C07299=1229.702,-97.800,-36.392,179.567,5.287,149.048
C07300=1229.707,-98.050,-36.382,179.565,5.287,149.049
C07301=1229.712,-98.299,-36.370,179.563,5.287,149.049
C07302=1229.718,-98.549,-36.360,179.561,5.287,149.050
C07303=1229.723,-98.799,-36.350,179.558,5.287,149.051
C07304=1229.728,-99.048,-36.339,179.556,5.287,149.052
C07305=1229.733,-99.298,-36.328,179.553,5.286,149.052
C07306=1229.738,-99.548,-36.318,179.551,5.287,149.053
C07307=1229.743,-99.798,-36.307,179.548,5.286,149.054
C07308=1229.748,-100.048,-36.296,179.546,5.287,149.054
C07309=1229.755,-100.319,-36.285,179.544,5.286,149.055
C07310=1229.759,-100.589,-36.273,179.542,5.287,149.056
C07311=1229.765,-100.861,-36.262,179.538,5.287,149.057
C07312=1229.772,-101.131,-36.250,179.536,5.286,149.057
C07313=1229.777,-101.382,-36.239,179.534,5.287,149.058
C07314=1229.782,-101.631,-36.229,179.531,5.286,149.059
C07315=1229.787,-101.881,-36.218,179.529,5.286,149.060
C07316=1229.793,-102.130,-36.207,179.527,5.286,149.060
C07317=1229.797,-102.380,-36.197,179.525,5.286,149.061
C07318=1229.802,-102.630,-36.187,179.523,5.286,149.062
C07319=1229.807,-102.880,-36.177,179.520,5.286,149.062
C07320=1229.813,-103.129,-36.166,179.518,5.286,149.063
C07321=1229.818,-103.379,-36.155,179.515,5.286,149.064
C07322=1229.823,-103.629,-36.145,179.513,5.286,149.064
C07323=1229.828,-103.879,-36.134,179.510,5.286,149.065
C07324=1229.834,-104.129,-36.124,179.508,5.286,149.066
C07325=1229.839,-104.377,-36.113,179.506,5.286,149.067
C07326=1229.844,-104.628,-36.103,179.503,5.286,149.067
C07327=1229.850,-104.877,-36.092,179.501,5.286,149.068
C07328=1229.855,-105.127,-36.082,179.499,5.286,149.069
C07329=1229.860,-105.377,-36.072,179.496,5.286,149.069
C07330=1229.865,-105.627,-36.061,179.494,5.286,149.070
C07331=1229.870,-105.876,-36.051,179.492,5.285,149.071
C07332=1229.875,-106.126,-36.040,179.490,5.285,149.071
C07333=1229.880,-106.376,-36.030,179.487,5.285,149.072
C07334=1229.886,-106.625,-36.020,179.485,5.285,149.073
C07335=1229.891,-106.875,-36.009,179.483,5.286,149.073
C07336=1229.897,-107.125,-35.999,179.480,5.285,149.074
C07337=1229.902,-107.375,-35.988,179.478,5.286,149.075
C07338=1229.907,-107.625,-35.978,179.475,5.285,149.076
C07339=1229.913,-107.874,-35.968,179.473,5.286,149.076
C07340=1229.917,-108.124,-35.957,179.471,5.285,149.077
C07341=1229.922,-108.373,-35.947,179.468,5.286,149.078
C07342=1229.927,-108.623,-35.937,179.466,5.285,149.078
C07343=1229.933,-108.873,-35.926,179.464,5.285,149.079
C07344=1229.939,-109.123,-35.916,179.462,5.285,149.080
C07345=1229.944,-109.373,-35.906,179.459,5.285,149.080
C07346=1229.948,-109.622,-35.896,179.457,5.285,149.081
C07347=1229.953,-109.872,-35.885,179.455,5.285,149.082
C07348=1229.959,-110.122,-35.875,179.453,5.285,149.082
C07349=1229.965,-110.371,-35.865,179.450,5.285,149.083
C07350=1229.970,-110.622,-35.854,179.448,5.285,149.084
C07351=1229.975,-110.871,-35.845,179.445,5.285,149.085
C07352=1229.980,-111.120,-35.835,179.443,5.285,149.085
C07353=1229.985,-111.371,-35.824,179.441,5.284,149.086
C07354=1229.991,-111.620,-35.814,179.439,5.285,149.087
C07355=1229.996,-111.870,-35.804,179.436,5.284,149.087
C07356=1230.001,-112.120,-35.794,179.434,5.285,149.088
C07357=1230.006,-112.369,-35.783,179.431,5.284,149.089
C07358=1230.011,-112.619,-35.773,179.429,5.285,149.089
C07359=1230.017,-112.869,-35.763,179.427,5.284,149.090
C07360=1230.022,-113.118,-35.752,179.424,5.285,149.091
C07361=1230.027,-113.368,-35.742,179.422,5.285,149.092
C07362=1230.032,-113.618,-35.732,179.420,5.285,149.092
C07363=1230.038,-113.867,-35.722,179.418,5.285,149.093
C07364=1230.044,-114.118,-35.712,179.415,5.284,149.093
C07365=1230.048,-114.368,-35.702,179.413,5.284,149.094
C07366=1230.054,-114.617,-35.692,179.411,5.284,149.095
C07367=1230.059,-114.867,-35.682,179.409,5.284,149.096
C07368=1230.064,-115.117,-35.671,179.406,5.284,149.096
C07369=1230.069,-115.366,-35.662,179.404,5.284,149.097
C07370=1230.075,-115.616,-35.652,179.401,5.284,149.098
C07371=1230.080,-115.866,-35.641,179.399,5.284,149.098
C07372=1230.085,-116.115,-35.631,179.397,5.284,149.099
C07373=1230.090,-116.365,-35.622,179.395,5.284,149.100
C07374=1230.095,-116.616,-35.611,179.393,5.284,149.100
C07375=1230.100,-116.865,-35.602,179.390,5.284,149.101
C07376=1230.106,-117.114,-35.592,179.388,5.284,149.102
C07377=1230.111,-117.364,-35.581,179.385,5.284,149.103
C07378=1230.116,-117.614,-35.571,179.383,5.284,149.103
C07379=1230.122,-117.864,-35.562,179.380,5.284,149.104
C07380=1230.127,-118.114,-35.552,179.379,5.284,149.104
C07381=1230.132,-118.363,-35.542,179.376,5.283,149.105
C07382=1230.137,-118.613,-35.532,179.374,5.284,149.106
C07383=1230.143,-118.863,-35.521,179.372,5.284,149.107
C07384=1230.148,-119.112,-35.512,179.369,5.284,149.107
C07385=1230.153,-119.363,-35.502,179.367,5.284,149.108
C07386=1230.158,-119.612,-35.492,179.364,5.284,149.109
C07387=1230.163,-119.861,-35.482,179.362,5.284,149.109
C07388=1230.169,-120.111,-35.472,179.360,5.283,149.110
C07389=1230.174,-120.362,-35.462,179.358,5.283,149.111
C07390=1230.179,-120.611,-35.452,179.355,5.283,149.111
C07391=1230.185,-120.861,-35.442,179.353,5.283,149.112
C07392=1230.190,-121.110,-35.433,179.351,5.284,149.113
C07393=1230.195,-121.360,-35.423,179.349,5.283,149.114
C07394=1230.200,-121.610,-35.412,179.346,5.284,149.114
C07395=1230.205,-121.859,-35.403,179.344,5.283,149.115
C07396=1230.211,-122.110,-35.393,179.342,5.283,149.115
C07397=1230.216,-122.359,-35.384,179.339,5.283,149.116
C07398=1230.221,-122.609,-35.373,179.337,5.283,149.117
C07399=1230.226,-122.859,-35.364,179.335,5.283,149.118
C07400=1230.232,-123.109,-35.354,179.333,5.283,149.118
C07401=1230.237,-123.358,-35.344,179.331,5.284,149.119
C07402=1230.243,-123.608,-35.335,179.328,5.283,149.120
C07403=1230.248,-123.858,-35.324,179.326,5.283,149.120
C07404=1230.252,-124.107,-35.315,179.324,5.283,149.121
C07405=1230.258,-124.358,-35.305,179.321,5.283,149.122
C07406=1230.263,-124.607,-35.296,179.319,5.283,149.122
C07407=1230.269,-124.856,-35.285,179.317,5.283,149.123
C07408=1230.273,-125.107,-35.276,179.314,5.283,149.124
C07409=1230.279,-125.356,-35.266,179.312,5.283,149.125
C07410=1230.284,-125.606,-35.256,179.310,5.283,149.125
C07411=1230.290,-125.856,-35.247,179.308,5.283,149.126
C07412=1230.295,-126.105,-35.237,179.306,5.283,149.126
C07413=1229.874,-126.116,-35.273,179.301,5.287,149.129
C07414=1229.868,-125.866,-35.282,179.303,5.286,149.128
C07415=1229.863,-125.617,-35.292,179.305,5.286,149.127
C07416=1229.857,-125.367,-35.302,179.308,5.286,149.126
C07417=1229.852,-125.117,-35.311,179.310,5.286,149.126
C07418=1229.846,-124.868,-35.321,179.313,5.286,149.125
C07419=1229.842,-124.617,-35.331,179.314,5.286,149.125
C07420=1229.836,-124.368,-35.341,179.317,5.287,149.124
C07421=1229.831,-124.118,-35.351,179.319,5.286,149.123
C07422=1229.826,-123.868,-35.360,179.322,5.287,149.122
C07423=1229.821,-123.619,-35.370,179.324,5.286,149.122
C07424=1229.816,-123.369,-35.380,179.326,5.286,149.121
C07425=1229.810,-123.119,-35.389,179.328,5.287,149.120
C07426=1229.805,-122.869,-35.399,179.330,5.286,149.120
C07427=1229.799,-122.620,-35.409,179.333,5.287,149.119
C07428=1229.794,-122.370,-35.418,179.335,5.286,149.118
C07429=1229.789,-122.120,-35.429,179.338,5.287,149.118
C07430=1229.784,-121.871,-35.439,179.340,5.286,149.117
C07431=1229.778,-121.620,-35.448,179.342,5.287,149.116
C07432=1229.773,-121.371,-35.458,179.345,5.287,149.115
C07433=1229.769,-121.121,-35.468,179.346,5.287,149.115
C07434=1229.763,-120.871,-35.478,179.349,5.287,149.114
C07435=1229.758,-120.622,-35.487,179.351,5.287,149.114
C07436=1229.752,-120.372,-35.498,179.354,5.287,149.113
C07437=1229.747,-120.122,-35.508,179.356,5.287,149.112
C07438=1229.742,-119.872,-35.518,179.358,5.287,149.111
C07439=1229.736,-119.622,-35.527,179.360,5.287,149.111
C07440=1229.732,-119.373,-35.537,179.363,5.287,149.110
C07441=1229.726,-119.124,-35.547,179.365,5.287,149.109
C07442=1229.721,-118.873,-35.558,179.367,5.288,149.109
C07443=1229.716,-118.623,-35.567,179.370,5.287,149.108
C07444=1229.710,-118.374,-35.577,179.372,5.287,149.107
C07445=1229.705,-118.124,-35.587,179.374,5.287,149.107
C07446=1229.700,-117.874,-35.597,179.376,5.287,149.106
C07447=1229.695,-117.625,-35.607,179.379,5.287,149.105
C07448=1229.689,-117.375,-35.617,179.381,5.287,149.105
C07449=1229.685,-117.125,-35.627,179.383,5.288,149.104
C07450=1229.679,-116.875,-35.637,179.385,5.287,149.103
C07451=1229.673,-116.626,-35.647,179.388,5.288,149.103
C07452=1229.668,-116.376,-35.657,179.390,5.287,149.102
C07453=1229.663,-116.126,-35.667,179.393,5.288,149.101
C07454=1229.658,-115.877,-35.677,179.395,5.287,149.100
C07455=1229.653,-115.627,-35.686,179.397,5.287,149.100
C07456=1229.648,-115.377,-35.697,179.399,5.288,149.099
C07457=1229.642,-115.127,-35.707,179.401,5.287,149.098
C07458=1229.637,-114.878,-35.717,179.404,5.288,149.098
C07459=1229.632,-114.628,-35.727,179.406,5.288,149.097
C07460=1229.627,-114.378,-35.738,179.409,5.288,149.096
C07461=1229.621,-114.128,-35.748,179.411,5.288,149.096
C07462=1229.616,-113.878,-35.758,179.414,5.288,149.095
C07463=1229.611,-113.629,-35.768,179.416,5.288,149.094
C07464=1229.606,-113.379,-35.778,179.418,5.288,149.093
C07465=1229.600,-113.129,-35.788,179.420,5.288,149.093
C07466=1229.595,-112.879,-35.798,179.422,5.288,149.092
C07467=1229.590,-112.630,-35.808,179.425,5.288,149.092
C07468=1229.584,-112.380,-35.818,179.427,5.288,149.091
C07469=1229.579,-112.130,-35.829,179.430,5.288,149.090
C07470=1229.574,-111.880,-35.839,179.432,5.288,149.089
C07471=1229.569,-111.631,-35.849,179.434,5.288,149.089
C07472=1229.564,-111.381,-35.859,179.436,5.288,149.088
C07473=1229.558,-111.131,-35.869,179.439,5.288,149.087
C07474=1229.553,-110.881,-35.880,179.441,5.288,149.087
C07475=1229.548,-110.632,-35.890,179.443,5.289,149.086
C07476=1229.543,-110.382,-35.900,179.445,5.288,149.085
C07477=1229.538,-110.132,-35.910,179.448,5.288,149.085
C07478=1229.532,-109.883,-35.920,179.450,5.288,149.084
C07479=1229.527,-109.633,-35.931,179.452,5.288,149.083
C07480=1229.522,-109.383,-35.941,179.455,5.289,149.082
C07481=1229.517,-109.134,-35.951,179.457,5.288,149.082
C07482=1229.512,-108.883,-35.961,179.460,5.289,149.081
C07483=1229.506,-108.634,-35.972,179.462,5.288,149.080
C07484=1229.500,-108.384,-35.982,179.465,5.289,149.080
C07485=1229.496,-108.135,-35.993,179.467,5.288,149.079
C07486=1229.490,-107.885,-36.003,179.469,5.289,149.078
C07487=1229.485,-107.635,-36.014,179.471,5.289,149.078
C07488=1229.480,-107.386,-36.023,179.474,5.289,149.077
C07489=1229.475,-107.136,-36.034,179.476,5.289,149.076
C07490=1229.470,-106.886,-36.044,179.478,5.289,149.076
C07491=1229.464,-106.636,-36.054,179.480,5.289,149.075
C07492=1229.459,-106.386,-36.065,179.483,5.289,149.074
C07493=1229.454,-106.137,-36.075,179.485,5.289,149.073
C07494=1229.448,-105.887,-36.085,179.487,5.289,149.073
C07495=1229.443,-105.637,-36.097,179.490,5.289,149.072
C07496=1229.438,-105.388,-36.106,179.492,5.289,149.071
C07497=1229.433,-105.138,-36.117,179.495,5.289,149.071
C07498=1229.428,-104.888,-36.127,179.496,5.289,149.070
C07499=1229.423,-104.638,-36.138,179.499,5.290,149.069
C07500=1229.417,-104.389,-36.148,179.501,5.289,149.069
C07501=1229.413,-104.139,-36.159,179.504,5.290,149.068
C07502=1229.407,-103.889,-36.169,179.506,5.289,149.067
C07503=1229.401,-103.640,-36.180,179.509,5.290,149.066
C07504=1229.396,-103.390,-36.190,179.511,5.289,149.066
C07505=1229.391,-103.140,-36.200,179.513,5.290,149.065
C07506=1229.386,-102.890,-36.212,179.515,5.289,149.064
C07507=1229.380,-102.641,-36.222,179.517,5.289,149.064
C07508=1229.375,-102.391,-36.232,179.520,5.289,149.063
C07509=1229.370,-102.141,-36.243,179.522,5.289,149.062
C07510=1229.365,-101.891,-36.253,179.525,5.290,149.062
C07511=1229.360,-101.642,-36.264,179.527,5.290,149.061
C07512=1229.355,-101.392,-36.275,179.529,5.290,149.060
C07513=1229.350,-101.142,-36.284,179.531,5.290,149.060
C07514=1229.344,-100.871,-36.297,179.534,5.290,149.059
C07515=1229.338,-100.600,-36.308,179.537,5.290,149.058
C07516=1229.333,-100.330,-36.319,179.539,5.290,149.057
C07517=1229.327,-100.058,-36.331,179.542,5.290,149.057
C07518=1229.322,-99.808,-36.342,179.544,5.290,149.056
C07519=1229.316,-99.559,-36.352,179.547,5.290,149.055
C07520=1229.311,-99.309,-36.363,179.549,5.290,149.054
C07521=1229.306,-99.059,-36.373,179.551,5.290,149.054
C07522=1229.301,-98.810,-36.385,179.554,5.290,149.053
C07523=1229.296,-98.560,-36.395,179.556,5.290,149.052
C07524=1229.291,-98.310,-36.405,179.558,5.290,149.052
C07525=1229.285,-98.061,-36.416,179.561,5.291,149.051
C07526=1229.280,-97.811,-36.427,179.563,5.291,149.050
C07527=1229.275,-97.561,-36.437,179.565,5.290,149.050
C07528=1229.270,-97.312,-36.448,179.567,5.291,149.049
C07529=1229.264,-97.062,-36.459,179.569,5.290,149.048
C07530=1229.259,-96.812,-36.469,179.572,5.291,149.047
C07531=1229.254,-96.563,-36.480,179.574,5.290,149.047
C07532=1229.249,-96.313,-36.491,179.577,5.291,149.046
C07533=1229.243,-96.063,-36.501,179.579,5.290,149.045
C07534=1229.238,-95.813,-36.513,179.582,5.291,149.045
C07535=1229.233,-95.563,-36.523,179.584,5.291,149.044
C07536=1229.228,-95.314,-36.534,179.586,5.291,149.043
C07537=1229.223,-95.064,-36.545,179.589,5.291,149.042
C07538=1229.218,-94.815,-36.556,179.591,5.291,149.042
C07539=1229.213,-94.565,-36.566,179.593,5.291,149.041
C07540=1229.207,-94.315,-36.576,179.596,5.291,149.040
C07541=1229.202,-94.065,-36.588,179.598,5.291,149.040
C07542=1229.196,-93.815,-36.599,179.601,5.291,149.039
C07543=1229.191,-93.566,-36.610,179.603,5.291,149.038
C07544=1229.186,-93.316,-36.620,179.606,5.291,149.037
C07545=1229.181,-93.067,-36.631,179.607,5.291,149.037
C07546=1229.176,-92.817,-36.642,179.610,5.292,149.036
C07547=1229.171,-92.567,-36.653,179.612,5.291,149.036
C07548=1229.166,-92.317,-36.663,179.615,5.292,149.035
C07549=1229.160,-92.067,-36.675,179.617,5.292,149.034
C07550=1229.155,-91.818,-36.686,179.619,5.292,149.033
C07551=1229.150,-91.568,-36.697,179.621,5.292,149.033
C07552=1229.145,-91.318,-36.707,179.624,5.292,149.032
C07553=1229.140,-91.069,-36.718,179.626,5.292,149.031
C07554=1229.135,-90.819,-36.729,179.629,5.292,149.031
C07555=1229.129,-90.570,-36.740,179.631,5.292,149.030
C07556=1229.124,-90.319,-36.751,179.634,5.292,149.029
C07557=1229.119,-90.070,-36.762,179.636,5.292,149.028
C07558=1229.114,-89.821,-36.773,179.638,5.292,149.028
C07559=1229.109,-89.571,-36.784,179.640,5.292,149.027
C07560=1229.103,-89.321,-36.796,179.643,5.292,149.026
C07561=1229.098,-89.071,-36.806,179.645,5.292,149.026
C07562=1229.093,-88.821,-36.817,179.648,5.293,149.025
C07563=1229.088,-88.571,-36.828,179.650,5.292,149.024
C07564=1229.082,-88.322,-36.839,179.653,5.293,149.023
C07565=1229.077,-88.072,-36.851,179.655,5.292,149.023
C07566=1229.072,-87.822,-36.861,179.657,5.293,149.022
C07567=1229.067,-87.573,-36.872,179.660,5.292,149.021
C07568=1229.061,-87.323,-36.884,179.662,5.293,149.021
C07569=1229.056,-87.073,-36.895,179.664,5.292,149.020
C07570=1229.051,-86.824,-36.905,179.666,5.293,149.019
C07571=1229.046,-86.574,-36.917,179.669,5.293,149.019
C07572=1229.041,-86.324,-36.928,179.671,5.293,149.018
C07573=1229.035,-86.075,-36.939,179.673,5.293,149.017
C07574=1229.031,-85.825,-36.950,179.675,5.293,149.017
C07575=1229.025,-85.575,-36.961,179.678,5.293,149.016
C07576=1229.020,-85.326,-36.972,179.680,5.293,149.015
C07577=1229.015,-85.076,-36.983,179.683,5.293,149.014
C07578=1229.010,-84.826,-36.994,179.686,5.294,149.014
C07579=1229.005,-84.576,-37.006,179.688,5.293,149.013
C07580=1228.999,-84.327,-37.017,179.690,5.294,149.012
C07581=1228.994,-84.077,-37.027,179.692,5.293,149.012
C07582=1228.989,-83.827,-37.039,179.695,5.294,149.011
C07583=1228.984,-83.578,-37.050,179.697,5.294,149.010
C07584=1228.979,-83.328,-37.062,179.700,5.294,149.010
C07585=1228.973,-83.078,-37.073,179.702,5.294,149.009
C07586=1228.968,-82.828,-37.084,179.705,5.294,149.008
C07587=1228.963,-82.579,-37.095,179.707,5.294,149.007
C07588=1228.958,-82.329,-37.107,179.709,5.294,149.007
C07589=1228.953,-82.080,-37.118,179.711,5.294,149.006
C07590=1228.948,-81.829,-37.129,179.714,5.294,149.005
C07591=1228.942,-81.580,-37.140,179.716,5.294,149.005
C07592=1228.937,-81.331,-37.151,179.719,5.294,149.004
C07593=1228.932,-81.081,-37.163,179.721,5.294,149.003
C07594=1228.927,-80.831,-37.175,179.724,5.295,149.002
C07595=1228.922,-80.582,-37.185,179.726,5.294,149.002
C07596=1228.916,-80.332,-37.197,179.728,5.295,149.001
C07597=1228.911,-80.082,-37.208,179.730,5.294,149.000
C07598=1228.906,-79.832,-37.220,179.733,5.295,149.000
C07599=1228.901,-79.583,-37.231,179.735,5.294,148.999
C07600=1228.896,-79.333,-37.242,179.738,5.295,148.998
C07601=1228.890,-79.083,-37.253,179.740,5.295,148.997
C07602=1228.886,-78.833,-37.265,179.743,5.295,148.997
C07603=1228.880,-78.583,-37.277,179.745,5.295,148.996
C07604=1228.875,-78.334,-37.287,179.747,5.295,148.995
C07605=1228.869,-78.084,-37.299,179.750,5.295,148.995
C07606=1228.865,-77.835,-37.311,179.752,5.295,148.994
C07607=1228.860,-77.585,-37.322,179.754,5.295,148.993
C07608=1228.855,-77.335,-37.334,179.757,5.295,148.992
C07609=1228.849,-77.086,-37.345,179.759,5.295,148.992
C07610=1228.844,-76.836,-37.356,179.762,5.295,148.991
C07611=1228.839,-76.586,-37.367,179.764,5.295,148.990
C07612=1228.834,-76.336,-37.379,179.766,5.296,148.990
C07613=1228.829,-76.087,-37.390,179.769,5.295,148.989
C07614=1228.823,-75.837,-37.402,179.771,5.296,148.988
C07615=1228.818,-75.588,-37.413,179.773,5.295,148.988
C07616=1228.813,-75.338,-37.425,179.776,5.296,148.987
C07617=1228.808,-75.088,-37.436,179.778,5.295,148.986
C07618=1228.802,-74.819,-37.449,179.781,5.296,148.985
C07619=1228.796,-74.548,-37.461,179.783,5.296,148.985
C07620=1228.791,-74.277,-37.474,179.786,5.296,148.984
C07621=1228.785,-74.007,-37.486,179.788,5.296,148.983
C07622=1228.780,-73.757,-37.498,179.791,5.297,148.983
C07623=1228.775,-73.507,-37.509,179.793,5.297,148.982
C07624=1228.769,-73.257,-37.521,179.796,5.297,148.981
C07625=1228.765,-73.008,-37.533,179.798,5.297,148.980
C07626=1228.760,-72.759,-37.545,179.800,5.297,148.980
C07627=1228.755,-72.509,-37.556,179.802,5.297,148.979
C07628=1228.749,-72.260,-37.568,179.805,5.297,148.978
C07629=1228.744,-72.010,-37.579,179.807,5.297,148.978
C07630=1228.739,-71.760,-37.591,179.810,5.297,148.977
C07631=1228.733,-71.510,-37.603,179.812,5.297,148.976
C07632=1228.729,-71.261,-37.614,179.815,5.298,148.975
C07633=1228.723,-71.011,-37.626,179.817,5.297,148.975
C07634=1228.718,-70.761,-37.637,179.819,5.298,148.974
C07635=1228.713,-70.511,-37.649,179.822,5.297,148.973
C07636=1228.707,-70.262,-37.661,179.824,5.298,148.973
C07637=1228.702,-70.012,-37.672,179.826,5.297,148.972
C07638=1228.697,-69.763,-37.685,179.829,5.298,148.971
C07639=1228.693,-69.513,-37.696,179.832,5.298,148.971
C07640=1228.687,-69.263,-37.708,179.834,5.298,148.970
C07641=1228.682,-69.013,-37.720,179.836,5.298,148.969
C07642=1228.677,-68.764,-37.731,179.838,5.298,148.968
C07643=1228.672,-68.514,-37.743,179.841,5.299,148.968
C07644=1228.666,-68.264,-37.755,179.843,5.298,148.967
C07645=1228.662,-68.015,-37.767,179.846,5.299,148.966
C07646=1228.656,-67.765,-37.779,179.848,5.298,148.966
C07647=1228.651,-67.515,-37.790,179.851,5.299,148.965
C07648=1228.646,-67.266,-37.801,179.853,5.299,148.964
C07649=1228.640,-67.016,-37.813,179.855,5.299,148.963
C07650=1228.635,-66.767,-37.826,179.858,5.299,148.963
C07651=1228.630,-66.517,-37.837,179.860,5.299,148.962
C07652=1228.625,-66.267,-37.849,179.862,5.299,148.961
C07653=1228.619,-66.017,-37.861,179.865,5.299,148.961
C07654=1228.615,-65.768,-37.872,179.868,5.300,148.960
C07655=1228.610,-65.518,-37.885,179.870,5.299,148.959
C07656=1228.604,-65.268,-37.897,179.872,5.300,148.959
C07657=1228.600,-65.019,-37.908,179.874,5.300,148.958
C07658=1228.594,-64.769,-37.920,179.877,5.300,148.957
C07659=1228.589,-64.520,-37.933,179.879,5.300,148.956
C07660=1228.584,-64.270,-37.944,179.882,5.300,148.956
C07661=1228.579,-64.020,-37.956,179.884,5.300,148.955
C07662=1228.574,-63.771,-37.968,179.887,5.300,148.954
C07663=1228.568,-63.521,-37.980,179.889,5.300,148.954
C07664=1228.564,-63.271,-37.991,179.891,5.300,148.953
C07665=1228.558,-63.022,-38.004,179.894,5.301,148.952
C07666=1228.553,-62.772,-38.016,179.897,5.300,148.951
C07667=1228.548,-62.522,-38.028,179.899,5.301,148.951
C07668=1228.543,-62.273,-38.040,179.901,5.300,148.950
C07669=1228.538,-62.023,-38.052,179.904,5.301,148.949
C07670=1228.532,-61.773,-38.064,179.906,5.300,148.948
C07671=1228.527,-61.524,-38.076,179.909,5.301,148.948
C07672=1228.522,-61.274,-38.088,179.911,5.301,148.947
C07673=1228.517,-61.024,-38.099,179.914,5.301,148.946
C07674=1228.512,-60.775,-38.112,179.916,5.301,148.946
C07675=1228.507,-60.525,-38.124,179.918,5.301,148.945
C07676=1228.501,-60.275,-38.136,179.921,5.302,148.944
C07677=1228.496,-60.026,-38.148,179.923,5.301,148.943
C07678=1228.491,-59.776,-38.160,179.926,5.302,148.943
C07679=1228.486,-59.527,-38.172,179.928,5.301,148.942
C07680=1228.481,-59.277,-38.184,179.931,5.302,148.941
C07681=1228.476,-59.027,-38.197,179.933,5.302,148.941
C07682=1228.470,-58.777,-38.209,179.935,5.302,148.940
C07683=1228.466,-58.528,-38.220,179.937,5.302,148.939
C07684=1228.461,-58.278,-38.233,179.940,5.302,148.939
C07685=1228.456,-58.028,-38.245,179.943,5.303,148.938
C07686=1228.450,-57.779,-38.257,179.945,5.302,148.937
C07687=1228.445,-57.529,-38.269,179.947,5.303,148.936
C07688=1228.440,-57.279,-38.282,179.950,5.302,148.936
C07689=1228.434,-57.029,-38.294,179.952,5.303,148.935
C07690=1228.430,-56.780,-38.306,179.954,5.303,148.934
C07691=1228.425,-56.530,-38.318,179.957,5.303,148.934
C07692=1228.420,-56.281,-38.330,179.960,5.304,148.933
C07693=1228.414,-56.031,-38.342,179.962,5.303,148.932
C07694=1228.409,-55.782,-38.355,179.964,5.304,148.931
C07695=1228.404,-55.532,-38.367,179.966,5.303,148.931
C07696=1228.399,-55.282,-38.380,179.969,5.304,148.930
C07697=1228.394,-55.032,-38.391,179.971,5.304,148.929
C07698=1228.388,-54.783,-38.404,179.974,5.304,148.929
C07699=1228.384,-54.534,-38.416,179.976,5.304,148.928
C07700=1228.379,-54.284,-38.428,179.979,5.304,148.927
C07701=1228.374,-54.034,-38.441,179.981,5.305,148.927
C07702=1228.368,-53.784,-38.452,179.983,5.304,148.926
C07703=1228.363,-53.535,-38.465,179.986,5.305,148.925
C07704=1228.358,-53.285,-38.477,179.988,5.304,148.924
C07705=1228.353,-53.035,-38.490,179.991,5.305,148.924
C07706=1228.348,-52.786,-38.502,179.993,5.305,148.923
C07707=1228.342,-52.536,-38.514,179.996,5.305,148.922
C07708=1228.337,-52.287,-38.527,179.998,5.306,148.922
C07709=1228.332,-52.037,-38.540,-180.000,5.305,148.921
C07710=1228.327,-51.787,-38.551,-179.997,5.306,148.920
C07711=1228.322,-51.537,-38.564,-179.995,5.305,148.920
C07712=1228.317,-51.287,-38.576,-179.992,5.306,148.919
C07713=1228.312,-51.038,-38.589,-179.990,5.306,148.918
C07714=1228.307,-50.789,-38.602,-179.988,5.306,148.917
C07715=1228.301,-50.539,-38.613,-179.985,5.306,148.917
C07716=1228.296,-50.290,-38.626,-179.983,5.306,148.916
C07717=1228.292,-50.040,-38.639,-179.980,5.307,148.915
C07718=1228.286,-49.790,-38.651,-179.978,5.306,148.915
C07719=1228.281,-49.540,-38.663,-179.975,5.307,148.914
C07720=1228.276,-49.291,-38.676,-179.973,5.307,148.913
C07721=1228.271,-49.042,-38.689,-179.971,5.307,148.912
C07722=1228.265,-48.771,-38.702,-179.967,5.307,148.912
C07723=1228.260,-48.501,-38.716,-179.965,5.308,148.911
C07724=1228.254,-48.232,-38.729,-179.963,5.307,148.910
C07725=1228.249,-47.962,-38.742,-179.960,5.308,148.909
C07726=1228.244,-47.713,-38.755,-179.957,5.308,148.909
C07727=1228.239,-47.463,-38.767,-179.955,5.308,148.908
C07728=1228.234,-47.213,-38.780,-179.953,5.308,148.907
C07729=1228.229,-46.963,-38.792,-179.951,5.308,148.907
C07730=1228.223,-46.714,-38.805,-179.948,5.309,148.906
C07731=1228.218,-46.464,-38.818,-179.946,5.308,148.905
C07732=1228.212,-46.215,-38.831,-179.943,5.308,148.904
C07733=1228.208,-45.965,-38.844,-179.940,5.309,148.904
C07734=1228.203,-45.715,-38.855,-179.938,5.308,148.903
C07735=1228.197,-45.466,-38.868,-179.935,5.309,148.902
C07736=1228.192,-45.216,-38.881,-179.933,5.309,148.901
C07737=1228.188,-44.966,-38.894,-179.930,5.309,148.901
C07738=1228.183,-44.717,-38.906,-179.928,5.310,148.900
C07739=1228.177,-44.467,-38.919,-179.926,5.309,148.899
C07740=1228.171,-44.218,-38.931,-179.923,5.310,148.899
C07741=1228.167,-43.967,-38.944,-179.921,5.309,148.898
C07742=1228.162,-43.718,-38.957,-179.918,5.310,148.897
C07743=1228.157,-43.469,-38.969,-179.916,5.310,148.897
C07744=1228.151,-43.220,-38.982,-179.914,5.310,148.896
C07745=1228.147,-42.970,-38.995,-179.911,5.311,148.895
C07746=1228.141,-42.720,-39.008,-179.909,5.310,148.894
C07747=1228.136,-42.471,-39.021,-179.906,5.311,148.894
C07748=1228.131,-42.221,-39.034,-179.903,5.311,148.893
C07749=1228.126,-41.971,-39.046,-179.901,5.311,148.892
C07750=1228.121,-41.721,-39.058,-179.899,5.311,148.892
C07751=1228.116,-41.472,-39.071,-179.897,5.311,148.891
C07752=1228.110,-41.222,-39.084,-179.894,5.312,148.890
C07753=1228.105,-40.972,-39.097,-179.891,5.312,148.890
C07754=1228.100,-40.723,-39.110,-179.889,5.312,148.889
C07755=1228.096,-40.473,-39.123,-179.887,5.312,148.888
C07756=1228.090,-40.223,-39.136,-179.884,5.312,148.887
C07757=1228.085,-39.974,-39.148,-179.882,5.312,148.887
C07758=1228.080,-39.724,-39.161,-179.879,5.313,148.886
C07759=1228.075,-39.475,-39.174,-179.877,5.313,148.885
C07760=1228.070,-39.225,-39.187,-179.874,5.313,148.885
C07761=1228.064,-38.976,-39.200,-179.872,5.313,148.884
C07762=1228.060,-38.726,-39.213,-179.870,5.313,148.883
C07763=1228.054,-38.476,-39.225,-179.867,5.314,148.883
C07764=1228.049,-38.227,-39.238,-179.865,5.313,148.882
C07765=1228.044,-37.977,-39.252,-179.862,5.314,148.881
C07766=1228.039,-37.727,-39.264,-179.860,5.314,148.880
C07767=1228.034,-37.478,-39.277,-179.857,5.314,148.880
C07768=1228.029,-37.228,-39.290,-179.855,5.315,148.879
C07769=1228.023,-36.979,-39.303,-179.853,5.314,148.878
C07770=1228.019,-36.728,-39.316,-179.850,5.315,148.878
C07771=1228.014,-36.480,-39.329,-179.847,5.315,148.877
C07772=1228.008,-36.230,-39.342,-179.845,5.315,148.876
C07773=1228.004,-35.980,-39.355,-179.843,5.315,148.876
C07774=1227.999,-35.731,-39.368,-179.841,5.315,148.875
C07775=1227.993,-35.481,-39.381,-179.838,5.316,148.874
C07776=1227.988,-35.231,-39.394,-179.835,5.316,148.873
C07777=1227.983,-34.982,-39.407,-179.833,5.315,148.873
C07778=1227.977,-34.732,-39.420,-179.830,5.316,148.872
C07779=1227.973,-34.482,-39.433,-179.828,5.316,148.871
C07780=1227.968,-34.234,-39.446,-179.825,5.316,148.870
C07781=1227.963,-33.983,-39.460,-179.823,5.317,148.870
C07782=1227.957,-33.734,-39.472,-179.821,5.316,148.869
C07783=1227.952,-33.485,-39.485,-179.818,5.317,148.868
C07784=1227.947,-33.234,-39.499,-179.815,5.317,148.868
C07785=1227.942,-32.985,-39.511,-179.813,5.317,148.867
C07786=1227.937,-32.735,-39.525,-179.810,5.317,148.866
C07787=1227.932,-32.486,-39.538,-179.808,5.317,148.866
C07788=1227.927,-32.236,-39.551,-179.806,5.318,148.865
C07789=1227.921,-31.986,-39.564,-179.803,5.318,148.864
C07790=1227.917,-31.738,-39.577,-179.801,5.318,148.863
C07791=1227.911,-31.487,-39.591,-179.798,5.318,148.863
C07792=1227.906,-31.238,-39.604,-179.796,5.319,148.862
C07793=1227.902,-30.988,-39.617,-179.794,5.318,148.861
C07794=1227.896,-30.738,-39.630,-179.791,5.319,148.861
C07795=1227.892,-30.489,-39.643,-179.789,5.319,148.860
C07796=1227.886,-30.239,-39.657,-179.786,5.319,148.859
C07797=1227.881,-29.990,-39.669,-179.783,5.320,148.859
C07798=1227.876,-29.741,-39.683,-179.781,5.319,148.858
C07799=1227.871,-29.491,-39.696,-179.779,5.320,148.857
C07800=1227.866,-29.241,-39.709,-179.776,5.320,148.856
C07801=1227.860,-28.991,-39.722,-179.774,5.320,148.856
C07802=1227.856,-28.742,-39.736,-179.771,5.321,148.855
C07803=1227.850,-28.492,-39.749,-179.769,5.321,148.854
C07804=1227.846,-28.242,-39.762,-179.767,5.321,148.854
C07805=1227.840,-27.993,-39.776,-179.764,5.321,148.853
C07806=1227.836,-27.743,-39.789,-179.762,5.321,148.852
C07807=1227.830,-27.494,-39.802,-179.759,5.321,148.852
C07808=1227.825,-27.244,-39.816,-179.757,5.322,148.851
C07809=1227.820,-26.994,-39.829,-179.754,5.322,148.850
C07810=1227.815,-26.745,-39.843,-179.752,5.322,148.849
C07811=1227.810,-26.495,-39.856,-179.749,5.323,148.849
C07812=1227.805,-26.245,-39.869,-179.747,5.322,148.848
C07813=1227.799,-25.996,-39.883,-179.744,5.323,148.847
C07814=1227.795,-25.746,-39.896,-179.742,5.323,148.847
C07815=1227.789,-25.497,-39.909,-179.740,5.323,148.846
C07816=1227.785,-25.247,-39.923,-179.737,5.323,148.845
C07817=1227.779,-24.998,-39.936,-179.734,5.324,148.845
C07818=1227.775,-24.748,-39.950,-179.732,5.324,148.844
C07819=1227.769,-24.499,-39.963,-179.730,5.324,148.843
C07820=1227.765,-24.249,-39.976,-179.727,5.325,148.843
C07821=1227.759,-24.000,-39.990,-179.725,5.324,148.842
C07822=1227.754,-23.750,-40.004,-179.722,5.325,148.841
C07823=1227.749,-23.501,-40.017,-179.719,5.325,148.840
C07824=1227.744,-23.251,-40.031,-179.717,5.325,148.840
C07825=1227.739,-23.001,-40.044,-179.714,5.325,148.839
C07826=1227.733,-22.732,-40.058,-179.712,5.326,148.838
C07827=1227.728,-22.463,-40.073,-179.710,5.325,148.837
C07828=1227.723,-22.193,-40.087,-179.707,5.326,148.837
C07829=1227.717,-21.924,-40.102,-179.704,5.326,148.836
C07830=1227.712,-21.675,-40.116,-179.701,5.327,148.835
C07831=1227.707,-21.425,-40.129,-179.699,5.326,148.834
C07832=1227.702,-21.176,-40.143,-179.696,5.327,148.834
C07833=1227.696,-20.925,-40.156,-179.694,5.327,148.833
C07834=1227.692,-20.677,-40.170,-179.692,5.327,148.832
C07835=1227.686,-20.426,-40.183,-179.689,5.327,148.832
C07836=1227.681,-20.177,-40.198,-179.686,5.328,148.831
C07837=1227.676,-19.927,-40.210,-179.684,5.328,148.830
C07838=1227.671,-19.678,-40.224,-179.682,5.328,148.830
C07839=1227.666,-19.429,-40.238,-179.679,5.329,148.829
C07840=1227.661,-19.179,-40.251,-179.677,5.328,148.828
C07841=1227.656,-18.929,-40.266,-179.674,5.329,148.827
C07842=1227.650,-18.679,-40.279,-179.671,5.329,148.827
C07843=1227.646,-18.430,-40.292,-179.669,5.329,148.826
C07844=1227.641,-18.181,-40.306,-179.667,5.330,148.825
C07845=1227.635,-17.930,-40.320,-179.664,5.330,148.825
C07846=1227.631,-17.681,-40.334,-179.662,5.330,148.824
C07847=1227.626,-17.432,-40.348,-179.659,5.330,148.823
C07848=1227.620,-17.182,-40.361,-179.657,5.331,148.823
C07849=1227.615,-16.933,-40.375,-179.655,5.330,148.822
C07850=1227.611,-16.683,-40.389,-179.652,5.331,148.821
C07851=1227.605,-16.433,-40.402,-179.649,5.332,148.821
C07852=1227.600,-16.184,-40.416,-179.647,5.331,148.820
C07853=1227.596,-15.935,-40.430,-179.645,5.332,148.819
C07854=1227.590,-15.684,-40.443,-179.642,5.332,148.818
C07855=1227.585,-15.435,-40.457,-179.640,5.332,148.818
C07856=1227.580,-15.186,-40.472,-179.637,5.332,148.817
C07857=1227.576,-14.936,-40.485,-179.635,5.333,148.816
C07858=1227.570,-14.686,-40.498,-179.632,5.333,148.816
C07859=1227.565,-14.437,-40.513,-179.630,5.333,148.815
C07860=1227.560,-14.187,-40.527,-179.627,5.334,148.814
C07861=1227.554,-13.938,-40.541,-179.625,5.333,148.814
C07862=1227.550,-13.688,-40.554,-179.622,5.334,148.813
C07863=1227.545,-13.438,-40.568,-179.620,5.334,148.812
C07864=1227.539,-13.189,-40.582,-179.617,5.335,148.811
C07865=1227.534,-12.940,-40.596,-179.615,5.335,148.811
C07866=1227.530,-12.690,-40.609,-179.612,5.335,148.810
C07867=1227.524,-12.441,-40.623,-179.610,5.336,148.809
C07868=1227.519,-12.191,-40.638,-179.608,5.335,148.809
C07869=1227.514,-11.941,-40.652,-179.605,5.336,148.808
C07870=1227.509,-11.691,-40.666,-179.602,5.336,148.807
C07871=1227.504,-11.442,-40.679,-179.600,5.336,148.807
C07872=1227.499,-11.192,-40.693,-179.598,5.337,148.806
C07873=1227.494,-10.943,-40.707,-179.595,5.337,148.805
C07874=1227.489,-10.694,-40.721,-179.593,5.337,148.805
C07875=1227.484,-10.444,-40.735,-179.590,5.337,148.804
C07876=1227.479,-10.194,-40.750,-179.587,5.338,148.803
C07877=1227.474,-9.945,-40.764,-179.585,5.338,148.802
C07878=1227.468,-9.696,-40.778,-179.583,5.338,148.802
C07879=1227.464,-9.446,-40.791,-179.580,5.339,148.801
C07880=1227.459,-9.196,-40.805,-179.577,5.339,148.800
C07881=1227.454,-8.946,-40.819,-179.575,5.339,148.800
C07882=1227.448,-8.697,-40.833,-179.573,5.339,148.799
C07883=1227.443,-8.447,-40.848,-179.570,5.340,148.798
C07884=1227.438,-8.198,-40.862,-179.568,5.340,148.798
C07885=1227.434,-7.948,-40.876,-179.565,5.340,148.797
C07886=1227.428,-7.699,-40.890,-179.563,5.341,148.796
C07887=1227.423,-7.449,-40.904,-179.560,5.341,148.796
C07888=1227.419,-7.200,-40.918,-179.558,5.341,148.795
C07889=1227.414,-6.950,-40.932,-179.555,5.341,148.794
C07890=1227.409,-6.700,-40.947,-179.553,5.342,148.793
C07891=1227.403,-6.451,-40.961,-179.551,5.342,148.793
C07892=1227.398,-6.202,-40.975,-179.548,5.342,148.792
C07893=1227.393,-5.952,-40.989,-179.545,5.343,148.791
C07894=1227.388,-5.702,-41.003,-179.543,5.343,148.791
C07895=1227.383,-5.453,-41.018,-179.541,5.343,148.790
C07896=1227.378,-5.204,-41.032,-179.538,5.343,148.789
C07897=1227.373,-4.954,-41.046,-179.535,5.344,148.789
C07898=1227.368,-4.704,-41.060,-179.533,5.344,148.788
C07899=1227.363,-4.454,-41.074,-179.530,5.344,148.787
C07900=1227.358,-4.205,-41.089,-179.528,5.345,148.787
C07901=1227.353,-3.956,-41.103,-179.525,5.345,148.786
C07902=1227.348,-3.706,-41.117,-179.523,5.345,148.785
C07903=1227.343,-3.456,-41.131,-179.520,5.345,148.785
C07904=1227.338,-3.207,-41.145,-179.518,5.346,148.784
C07905=1227.333,-2.957,-41.160,-179.516,5.346,148.783
C07906=1227.328,-2.707,-41.174,-179.513,5.346,148.782
C07907=1227.323,-2.459,-41.189,-179.510,5.347,148.782
C07908=1227.318,-2.209,-41.203,-179.508,5.347,148.781
C07909=1227.313,-1.959,-41.217,-179.506,5.347,148.780
C07910=1227.308,-1.710,-41.231,-179.503,5.347,148.780
C07911=1227.303,-1.460,-41.246,-179.500,5.348,148.779
C07912=1227.298,-1.210,-41.260,-179.498,5.348,148.778
C07913=1227.292,-0.961,-41.274,-179.496,5.348,148.778
C07914=1227.288,-0.712,-41.289,-179.493,5.349,148.777
C07915=1227.283,-0.462,-41.303,-179.490,5.349,148.776
C07916=1227.278,-0.213,-41.317,-179.488,5.349,148.776
C07917=1227.272,0.037,-41.332,-179.486,5.349,148.775
C07918=1227.267,0.287,-41.347,-179.483,5.350,148.774
C07919=1227.262,0.537,-41.361,-179.480,5.350,148.773
C07920=1227.257,0.786,-41.376,-179.478,5.350,148.773
C07921=1227.252,1.035,-41.390,-179.476,5.351,148.772
C07922=1227.247,1.285,-41.404,-179.473,5.351,148.771
C07923=1227.242,1.534,-41.418,-179.470,5.352,148.771
C07924=1227.237,1.783,-41.433,-179.468,5.351,148.770
C07925=1227.232,2.033,-41.448,-179.466,5.352,148.769
C07926=1227.227,2.283,-41.462,-179.463,5.352,148.769
C07927=1227.222,2.533,-41.477,-179.460,5.353,148.768
C07928=1227.217,2.782,-41.492,-179.458,5.353,148.767
C07929=1227.212,3.032,-41.506,-179.455,5.353,148.767
C07930=1227.207,3.300,-41.522,-179.453,5.354,148.766
C07931=1227.202,3.569,-41.537,-179.450,5.354,148.765
C07932=1227.195,3.838,-41.553,-179.447,5.354,148.764
C07933=1227.190,4.107,-41.568,-179.444,5.355,148.764
C07934=1227.185,4.356,-41.583,-179.442,5.355,148.763
C07935=1227.180,4.606,-41.598,-179.440,5.355,148.762
C07936=1227.175,4.856,-41.612,-179.437,5.356,148.762
C07937=1227.170,5.105,-41.627,-179.434,5.356,148.761
C07938=1227.165,5.355,-41.642,-179.432,5.356,148.760
C07939=1227.160,5.604,-41.656,-179.430,5.357,148.759
C07940=1227.155,5.853,-41.671,-179.427,5.357,148.759
C07941=1227.150,6.103,-41.685,-179.424,5.358,148.758
C07942=1227.145,6.353,-41.700,-179.422,5.357,148.757
C07943=1227.140,6.602,-41.715,-179.420,5.358,148.757
C07944=1227.135,6.852,-41.729,-179.417,5.358,148.756
C07945=1227.131,7.101,-41.744,-179.414,5.359,148.755
C07946=1227.125,7.351,-41.759,-179.412,5.359,148.755
C07947=1227.120,7.601,-41.774,-179.410,5.359,148.754
C07948=1227.115,7.850,-41.789,-179.407,5.360,148.753
C07949=1227.110,8.100,-41.803,-179.404,5.360,148.753
C07950=1227.105,8.349,-41.818,-179.402,5.360,148.752
C07951=1227.100,8.599,-41.833,-179.400,5.360,148.751
C07952=1227.095,8.848,-41.848,-179.397,5.361,148.751
C07953=1227.090,9.098,-41.862,-179.394,5.361,148.750
C07954=1227.085,9.347,-41.878,-179.392,5.362,148.749
C07955=1227.080,9.597,-41.892,-179.389,5.362,148.748
C07956=1227.075,9.846,-41.907,-179.387,5.362,148.748
C07957=1227.070,10.096,-41.922,-179.384,5.363,148.747
C07958=1227.065,10.345,-41.937,-179.382,5.363,148.746
C07959=1227.060,10.595,-41.951,-179.379,5.363,148.746
C07960=1227.055,10.844,-41.967,-179.377,5.364,148.745
C07961=1227.050,11.094,-41.981,-179.374,5.364,148.744
C07962=1227.045,11.343,-41.996,-179.372,5.365,148.744
C07963=1227.039,11.593,-42.011,-179.370,5.365,148.743
C07964=1227.035,11.842,-42.026,-179.367,5.365,148.743
C07965=1227.030,12.092,-42.040,-179.365,5.366,148.742
C07966=1227.024,12.341,-42.056,-179.362,5.366,148.741
C07967=1227.019,12.591,-42.070,-179.359,5.367,148.741
C07968=1227.015,12.840,-42.085,-179.357,5.367,148.740
C07969=1227.009,13.089,-42.100,-179.355,5.367,148.739
C07970=1227.005,13.340,-42.115,-179.352,5.368,148.738
C07971=1227.000,13.589,-42.130,-179.349,5.368,148.738
C07972=1226.995,13.838,-42.146,-179.347,5.369,148.737
C07973=1226.990,14.088,-42.160,-179.345,5.368,148.736
C07974=1226.985,14.337,-42.176,-179.342,5.369,148.736
C07975=1226.980,14.587,-42.190,-179.339,5.370,148.735
C07976=1226.975,14.836,-42.205,-179.337,5.370,148.734
C07977=1226.970,15.085,-42.220,-179.335,5.370,148.734
C07978=1226.965,15.335,-42.235,-179.332,5.370,148.733
C07979=1226.959,15.585,-42.250,-179.329,5.371,148.732
C07980=1226.955,15.834,-42.265,-179.327,5.371,148.732
C07981=1226.949,16.084,-42.280,-179.324,5.372,148.731
C07982=1226.945,16.333,-42.295,-179.322,5.372,148.730
C07983=1226.940,16.583,-42.310,-179.319,5.372,148.730
C07984=1226.935,16.832,-42.326,-179.317,5.373,148.729
C07985=1226.930,17.082,-42.340,-179.314,5.373,148.728
C07986=1226.925,17.331,-42.356,-179.311,5.374,148.728
C07987=1226.920,17.580,-42.371,-179.309,5.374,148.727
C07988=1226.914,17.830,-42.386,-179.307,5.374,148.726
C07989=1226.910,18.079,-42.401,-179.304,5.375,148.725
C07990=1226.905,18.329,-42.417,-179.301,5.375,148.725
C07991=1226.900,18.578,-42.432,-179.299,5.376,148.724
C07992=1226.895,18.828,-42.447,-179.297,5.375,148.723
C07993=1226.890,19.078,-42.462,-179.294,5.376,148.723
C07994=1226.884,19.327,-42.477,-179.292,5.377,148.722
C07995=1226.880,19.576,-42.492,-179.289,5.377,148.722
C07996=1226.875,19.826,-42.508,-179.286,5.378,148.721
C07997=1226.870,20.075,-42.523,-179.284,5.378,148.720
C07998=1226.865,20.325,-42.538,-179.282,5.378,148.720
C07999=1226.860,20.574,-42.553,-179.279,5.379,148.719
C08000=1226.855,20.824,-42.569,-179.276,5.379,148.718
C08001=1226.850,21.073,-42.584,-179.274,5.380,148.718
C08002=1226.845,21.323,-42.599,-179.271,5.380,148.717
C08003=1226.840,21.572,-42.615,-179.269,5.380,148.716
C08004=1226.835,21.822,-42.629,-179.266,5.381,148.715
C08005=1226.829,22.071,-42.645,-179.264,5.381,148.715
C08006=1226.825,22.321,-42.660,-179.261,5.382,148.714
C08007=1226.820,22.571,-42.676,-179.259,5.382,148.713
C08008=1226.815,22.820,-42.691,-179.256,5.382,148.713
C08009=1226.810,23.069,-42.706,-179.254,5.383,148.712
C08010=1226.805,23.319,-42.722,-179.251,5.383,148.711
C08011=1226.800,23.568,-42.737,-179.249,5.384,148.711
C08012=1226.795,23.818,-42.753,-179.246,5.384,148.710
C08013=1226.790,24.067,-42.768,-179.243,5.385,148.709
C08014=1226.785,24.316,-42.784,-179.242,5.385,148.709
C08015=1226.780,24.566,-42.799,-179.239,5.385,148.708
C08016=1226.776,24.815,-42.815,-179.236,5.386,148.708
C08017=1226.770,25.065,-42.830,-179.234,5.386,148.707
C08018=1226.765,25.314,-42.846,-179.231,5.387,148.706
C08019=1226.760,25.563,-42.861,-179.228,5.388,148.705
C08020=1226.755,25.813,-42.877,-179.226,5.387,148.705
C08021=1226.750,26.063,-42.892,-179.224,5.388,148.704
C08022=1226.745,26.312,-42.907,-179.221,5.388,148.703
C08023=1226.740,26.561,-42.923,-179.218,5.389,148.703
C08024=1226.735,26.811,-42.939,-179.216,5.389,148.702
C08025=1226.731,27.061,-42.954,-179.213,5.390,148.701
C08026=1226.725,27.310,-42.969,-179.211,5.390,148.701
C08027=1226.720,27.559,-42.985,-179.208,5.390,148.700
C08028=1226.716,27.809,-43.000,-179.206,5.391,148.699
C08029=1226.710,28.059,-43.016,-179.203,5.391,148.699
C08030=1226.705,28.308,-43.031,-179.200,5.392,148.698
C08031=1226.701,28.558,-43.047,-179.198,5.393,148.698
C08032=1226.696,28.807,-43.062,-179.196,5.393,148.697
C08033=1226.690,29.057,-43.078,-179.194,5.393,148.696
C08034=1226.685,29.325,-43.095,-179.191,5.394,148.696
C08035=1226.680,29.593,-43.111,-179.188,5.394,148.695
C08036=1226.675,29.862,-43.129,-179.185,5.394,148.694
C08037=1226.669,30.131,-43.146,-179.183,5.395,148.693
C08038=1226.664,30.380,-43.161,-179.180,5.395,148.693
C08039=1226.659,30.630,-43.177,-179.177,5.396,148.692
C08040=1226.654,30.879,-43.192,-179.175,5.397,148.691
C08041=1226.649,31.129,-43.208,-179.172,5.397,148.691
C08042=1226.644,31.378,-43.224,-179.169,5.398,148.690
C08043=1226.639,31.628,-43.240,-179.167,5.397,148.689
C08044=1226.634,31.877,-43.256,-179.165,5.398,148.689
C08045=1226.629,32.126,-43.271,-179.162,5.399,148.688
C08046=1226.624,32.376,-43.287,-179.160,5.399,148.687
C08047=1226.619,32.626,-43.302,-179.157,5.400,148.687
C08048=1226.615,32.875,-43.319,-179.155,5.401,148.686
C08049=1226.609,33.125,-43.335,-179.152,5.401,148.685
C08050=1226.604,33.374,-43.350,-179.150,5.401,148.685
C08051=1226.600,33.624,-43.366,-179.147,5.401,148.684
C08052=1226.595,33.873,-43.382,-179.145,5.402,148.683
C08053=1226.589,34.122,-43.397,-179.142,5.402,148.683
C08054=1226.584,34.372,-43.413,-179.139,5.403,148.682
C08055=1226.579,34.621,-43.430,-179.137,5.404,148.681
C08056=1226.575,34.871,-43.445,-179.134,5.404,148.681
C08057=1226.570,35.120,-43.461,-179.132,5.404,148.680
C08058=1226.565,35.369,-43.476,-179.130,5.405,148.679
C08059=1226.560,35.619,-43.493,-179.127,5.405,148.679
C08060=1226.555,35.868,-43.509,-179.124,5.406,148.678
C08061=1226.549,36.118,-43.524,-179.122,5.406,148.677
C08062=1226.545,36.367,-43.541,-179.119,5.407,148.677
C08063=1226.539,36.617,-43.556,-179.117,5.408,148.676
C08064=1226.535,36.867,-43.572,-179.114,5.408,148.675
C08065=1226.530,37.115,-43.588,-179.112,5.408,148.675
C08066=1226.526,37.365,-43.604,-179.109,5.408,148.674
C08067=1226.520,37.614,-43.620,-179.107,5.409,148.673
C08068=1226.515,37.863,-43.636,-179.104,5.410,148.673
C08069=1226.510,38.114,-43.652,-179.102,5.410,148.672
C08070=1226.505,38.362,-43.668,-179.099,5.411,148.672
C08071=1226.500,38.612,-43.684,-179.096,5.412,148.671
C08072=1226.495,38.861,-43.700,-179.094,5.412,148.670
C08073=1226.491,39.111,-43.716,-179.091,5.413,148.670
C08074=1226.485,39.361,-43.732,-179.089,5.412,148.669
C08075=1226.480,39.610,-43.748,-179.086,5.413,148.668
C08076=1226.475,39.860,-43.764,-179.084,5.413,148.668
C08077=1226.470,40.108,-43.780,-179.081,5.414,148.667
C08078=1226.465,40.359,-43.796,-179.079,5.415,148.666
C08079=1226.460,40.607,-43.813,-179.076,5.416,148.666
C08080=1226.456,40.857,-43.829,-179.074,5.416,148.665
C08081=1226.450,41.106,-43.845,-179.071,5.417,148.664
C08082=1226.446,41.356,-43.861,-179.068,5.417,148.664
C08083=1226.441,41.605,-43.877,-179.066,5.418,148.663
C08084=1226.436,41.855,-43.893,-179.064,5.418,148.662
C08085=1226.431,42.104,-43.909,-179.061,5.418,148.662
C08086=1226.426,42.354,-43.925,-179.058,5.419,148.661
C08087=1226.421,42.603,-43.942,-179.056,5.419,148.660
C08088=1226.416,42.852,-43.958,-179.053,5.420,148.660
C08089=1226.411,43.102,-43.974,-179.051,5.421,148.659
C08090=1226.407,43.351,-43.991,-179.048,5.421,148.659
C08091=1226.401,43.601,-44.006,-179.046,5.422,148.658
C08092=1226.397,43.850,-44.023,-179.043,5.422,148.657
C08093=1226.391,44.100,-44.039,-179.041,5.423,148.657
C08094=1226.386,44.349,-44.056,-179.038,5.423,148.656
C08095=1226.381,44.598,-44.072,-179.036,5.423,148.655
C08096=1226.376,44.848,-44.088,-179.033,5.424,148.655
C08097=1226.371,45.097,-44.104,-179.031,5.424,148.654
C08098=1226.367,45.346,-44.121,-179.028,5.425,148.653
C08099=1226.362,45.597,-44.137,-179.026,5.426,148.653
C08100=1226.357,45.845,-44.153,-179.023,5.426,148.652
C08101=1226.352,46.095,-44.169,-179.020,5.427,148.651
C08102=1226.347,46.344,-44.186,-179.018,5.428,148.651
C08103=1226.342,46.594,-44.203,-179.015,5.428,148.650
C08104=1226.337,46.843,-44.219,-179.013,5.429,148.649
C08105=1226.332,47.093,-44.235,-179.010,5.429,148.649
C08106=1226.327,47.342,-44.251,-179.008,5.430,148.648
C08107=1226.322,47.591,-44.268,-179.006,5.430,148.648
C08108=1226.317,47.841,-44.284,-179.003,5.430,148.647
C08109=1226.312,48.090,-44.300,-179.000,5.431,148.646
C08110=1226.307,48.340,-44.318,-178.998,5.432,148.646
C08111=1226.302,48.589,-44.334,-178.995,5.432,148.645
C08112=1226.297,48.839,-44.350,-178.993,5.433,148.644
C08113=1226.293,49.088,-44.366,-178.990,5.433,148.644
C08114=1226.288,49.337,-44.383,-178.988,5.434,148.643
C08115=1226.282,49.587,-44.400,-178.985,5.435,148.642
C08116=1226.277,49.836,-44.416,-178.982,5.435,148.642
C08117=1226.273,50.086,-44.432,-178.980,5.436,148.641
C08118=1226.268,50.335,-44.449,-178.977,5.436,148.640
C08119=1226.263,50.584,-44.465,-178.975,5.437,148.640
C08120=1226.258,50.834,-44.483,-178.972,5.438,148.639
C08121=1226.253,51.083,-44.499,-178.969,5.438,148.638
C08122=1226.248,51.333,-44.515,-178.968,5.438,148.638
C08123=1226.243,51.582,-44.531,-178.965,5.439,148.637
C08124=1226.238,51.831,-44.548,-178.962,5.439,148.637
C08125=1226.233,52.081,-44.565,-178.960,5.440,148.636
C08126=1226.229,52.330,-44.582,-178.957,5.441,148.635
C08127=1226.224,52.579,-44.598,-178.955,5.441,148.635
C08128=1226.218,52.829,-44.615,-178.952,5.442,148.634
C08129=1226.214,53.079,-44.631,-178.950,5.443,148.634
C08130=1226.209,53.328,-44.648,-178.947,5.443,148.633
C08131=1226.204,53.577,-44.664,-178.944,5.444,148.632
C08132=1226.199,53.827,-44.681,-178.942,5.444,148.632
C08133=1226.194,54.076,-44.698,-178.939,5.445,148.631
C08134=1226.189,54.325,-44.714,-178.937,5.445,148.630
C08135=1226.184,54.575,-44.732,-178.934,5.446,148.630
C08136=1226.179,54.824,-44.748,-178.932,5.447,148.629
C08137=1226.175,55.073,-44.765,-178.929,5.447,148.628
C08138=1226.169,55.342,-44.783,-178.927,5.448,148.628
C08139=1226.164,55.610,-44.801,-178.924,5.449,148.627
C08140=1226.158,55.880,-44.819,-178.921,5.449,148.626
C08141=1226.153,56.147,-44.837,-178.918,5.449,148.626
C08142=1226.148,56.397,-44.853,-178.916,5.450,148.625
C08143=1226.143,56.647,-44.871,-178.913,5.451,148.624
C08144=1226.138,56.895,-44.887,-178.911,5.451,148.624
C08145=1226.134,57.145,-44.904,-178.908,5.452,148.623
C08146=1226.128,57.395,-44.921,-178.905,5.453,148.622
C08147=1226.123,57.643,-44.937,-178.903,5.453,148.622
C08148=1226.118,57.893,-44.955,-178.900,5.454,148.621
C08149=1226.114,58.142,-44.972,-178.898,5.455,148.621
C08150=1226.110,58.392,-44.989,-178.895,5.455,148.620
C08151=1226.104,58.641,-45.005,-178.893,5.456,148.619
C08152=1226.099,58.890,-45.022,-178.890,5.456,148.619
C08153=1226.094,59.140,-45.039,-178.887,5.457,148.618
C08154=1226.090,59.389,-45.056,-178.885,5.458,148.617
C08155=1226.084,59.639,-45.073,-178.883,5.459,148.617
C08156=1226.079,59.888,-45.090,-178.880,5.459,148.616
C08157=1226.074,60.138,-45.107,-178.877,5.460,148.616
C08158=1226.070,60.387,-45.124,-178.875,5.460,148.615
C08159=1226.065,60.636,-45.141,-178.872,5.461,148.614
C08160=1226.060,60.885,-45.158,-178.870,5.461,148.614
C08161=1226.055,61.135,-45.175,-178.867,5.462,148.613
C08162=1226.050,61.385,-45.192,-178.865,5.463,148.612
C08163=1226.045,61.634,-45.208,-178.862,5.463,148.612
C08164=1226.040,61.883,-45.226,-178.860,5.464,148.611
C08165=1226.035,62.132,-45.243,-178.857,5.465,148.610
C08166=1226.030,62.382,-45.260,-178.854,5.465,148.610
C08167=1226.026,62.631,-45.277,-178.852,5.466,148.609
C08168=1226.020,62.881,-45.294,-178.849,5.467,148.609
C08169=1226.016,63.129,-45.311,-178.847,5.467,148.608
C08170=1226.010,63.379,-45.328,-178.844,5.468,148.607
C08171=1226.006,63.629,-45.345,-178.842,5.468,148.607
C08172=1226.001,63.878,-45.362,-178.839,5.469,148.606
C08173=1225.997,64.127,-45.380,-178.837,5.470,148.606
C08174=1225.991,64.377,-45.397,-178.834,5.471,148.605
C08175=1225.986,64.626,-45.414,-178.832,5.471,148.604
C08176=1225.981,64.875,-45.431,-178.829,5.472,148.604
C08177=1225.976,65.125,-45.448,-178.826,5.472,148.603
C08178=1225.972,65.374,-45.465,-178.824,5.473,148.603
C08179=1225.967,65.623,-45.483,-178.822,5.474,148.602
C08180=1225.962,65.873,-45.500,-178.819,5.474,148.601
C08181=1225.956,66.122,-45.517,-178.816,5.475,148.601
C08182=1225.952,66.371,-45.535,-178.814,5.476,148.600
C08183=1225.947,66.621,-45.551,-178.811,5.476,148.599
C08184=1225.942,66.870,-45.569,-178.809,5.477,148.599
C08185=1225.938,67.119,-45.586,-178.806,5.478,148.598
C08186=1225.932,67.369,-45.603,-178.804,5.478,148.597
C08187=1225.927,67.619,-45.620,-178.801,5.479,148.597
C08188=1225.923,67.868,-45.638,-178.798,5.479,148.596
C08189=1225.917,68.117,-45.655,-178.796,5.480,148.596
C08190=1225.912,68.366,-45.673,-178.794,5.481,148.595
C08191=1225.908,68.616,-45.689,-178.791,5.481,148.594
C08192=1225.903,68.865,-45.707,-178.788,5.482,148.594
C08193=1225.898,69.114,-45.725,-178.786,5.483,148.593
C08194=1225.893,69.364,-45.741,-178.784,5.484,148.593
C08195=1225.888,69.613,-45.759,-178.781,5.484,148.592
C08196=1225.883,69.863,-45.777,-178.778,5.485,148.591
C08197=1225.879,70.112,-45.794,-178.776,5.485,148.591
C08198=1225.874,70.362,-45.811,-178.773,5.486,148.590
C08199=1225.869,70.611,-45.829,-178.771,5.487,148.590
C08200=1225.864,70.860,-45.846,-178.768,5.487,148.589
C08201=1225.859,71.109,-45.863,-178.766,5.488,148.588
C08202=1225.854,71.359,-45.881,-178.763,5.489,148.588
C08203=1225.849,71.607,-45.898,-178.761,5.489,148.587
C08204=1225.844,71.857,-45.915,-178.758,5.491,148.586
C08205=1225.839,72.106,-45.933,-178.755,5.491,148.586
C08206=1225.834,72.356,-45.951,-178.752,5.492,148.585
C08207=1225.830,72.605,-45.968,-178.750,5.493,148.585
C08208=1225.825,72.854,-45.986,-178.748,5.494,148.584
C08209=1225.820,73.104,-46.003,-178.745,5.494,148.583
C08210=1225.815,73.353,-46.021,-178.742,5.495,148.583
C08211=1225.810,73.603,-46.038,-178.740,5.495,148.582
C08212=1225.805,73.852,-46.056,-178.737,5.496,148.581
C08213=1225.801,74.101,-46.074,-178.735,5.497,148.581
C08214=1225.795,74.351,-46.091,-178.732,5.497,148.580
C08215=1225.790,74.600,-46.109,-178.730,5.498,148.580
C08216=1225.786,74.849,-46.126,-178.727,5.499,148.579
C08217=1225.781,75.099,-46.144,-178.725,5.500,148.579
C08218=1225.776,75.348,-46.162,-178.722,5.500,148.578
C08219=1225.771,75.598,-46.179,-178.720,5.501,148.577
C08220=1225.766,75.847,-46.197,-178.717,5.501,148.577
C08221=1225.761,76.096,-46.215,-178.714,5.502,148.576
C08222=1225.757,76.345,-46.232,-178.712,5.504,148.576
C08223=1225.752,76.595,-46.250,-178.709,5.504,148.575
C08224=1225.747,76.844,-46.268,-178.707,5.505,148.574
C08225=1225.742,77.093,-46.286,-178.704,5.505,148.574
C08226=1225.737,77.343,-46.303,-178.702,5.506,148.573
C08227=1225.732,77.592,-46.321,-178.699,5.507,148.572
C08228=1225.728,77.841,-46.338,-178.697,5.508,148.572
C08229=1225.723,78.090,-46.356,-178.694,5.508,148.571
C08230=1225.717,78.340,-46.373,-178.692,5.509,148.571
C08231=1225.713,78.589,-46.391,-178.689,5.510,148.570
C08232=1225.708,78.838,-46.409,-178.686,5.510,148.569
C08233=1225.703,79.087,-46.427,-178.684,5.511,148.569
C08234=1225.698,79.338,-46.445,-178.682,5.512,148.568
C08235=1225.693,79.587,-46.463,-178.679,5.512,148.568
C08236=1225.688,79.836,-46.481,-178.676,5.514,148.567
C08237=1225.683,80.085,-46.499,-178.673,5.514,148.566
C08238=1225.678,80.335,-46.517,-178.671,5.515,148.566
C08239=1225.674,80.583,-46.534,-178.669,5.516,148.565
C08240=1225.669,80.833,-46.552,-178.666,5.517,148.565
C08241=1225.664,81.082,-46.570,-178.663,5.517,148.564
C08242=1225.659,81.351,-46.589,-178.661,5.518,148.563
C08243=1225.653,81.619,-46.609,-178.658,5.518,148.563
C08244=1225.648,81.887,-46.628,-178.655,5.520,148.562
C08245=1225.643,82.156,-46.647,-178.652,5.520,148.561
C08246=1225.638,82.405,-46.665,-178.650,5.521,148.561
C08247=1225.633,82.655,-46.683,-178.647,5.522,148.560
C08248=1225.628,82.904,-46.701,-178.645,5.522,148.560
C08249=1225.623,83.153,-46.719,-178.642,5.523,148.559
C08250=1225.618,83.402,-46.737,-178.640,5.524,148.559
C08251=1225.614,83.652,-46.755,-178.637,5.525,148.558
C08252=1225.609,83.901,-46.773,-178.634,5.526,148.557
C08253=1225.604,84.150,-46.791,-178.632,5.527,148.557
C08254=1225.599,84.400,-46.809,-178.629,5.528,148.556
C08255=1225.594,84.649,-46.827,-178.627,5.528,148.556
C08256=1225.589,84.898,-46.845,-178.624,5.529,148.555
C08257=1225.584,85.147,-46.863,-178.622,5.530,148.554
C08258=1225.580,85.397,-46.882,-178.619,5.530,148.554
C08259=1225.575,85.646,-46.899,-178.617,5.531,148.553
C08260=1225.570,85.895,-46.917,-178.614,5.532,148.552
C08261=1225.565,86.145,-46.935,-178.612,5.533,148.552
C08262=1225.560,86.394,-46.953,-178.609,5.534,148.551
C08263=1225.556,86.643,-46.971,-178.606,5.534,148.551
C08264=1225.551,86.893,-46.990,-178.604,5.535,148.550
C08265=1225.546,87.142,-47.008,-178.602,5.536,148.550
C08266=1225.541,87.391,-47.026,-178.599,5.537,148.549
C08267=1225.536,87.641,-47.044,-178.596,5.537,148.548
C08268=1225.531,87.890,-47.062,-178.594,5.538,148.548
C08269=1225.527,88.139,-47.081,-178.591,5.540,148.547
C08270=1225.522,88.388,-47.099,-178.588,5.540,148.547
C08271=1225.517,88.637,-47.117,-178.586,5.541,148.546
C08272=1225.512,88.887,-47.135,-178.584,5.542,148.546
C08273=1225.506,89.136,-47.154,-178.581,5.542,148.545
C08274=1225.502,89.386,-47.172,-178.578,5.543,148.544
C08275=1225.497,89.635,-47.190,-178.576,5.544,148.544
C08276=1225.493,89.884,-47.209,-178.573,5.545,148.543
C08277=1225.488,90.133,-47.227,-178.570,5.546,148.543
C08278=1225.483,90.383,-47.245,-178.568,5.546,148.542
C08279=1225.478,90.632,-47.264,-178.566,5.547,148.541
C08280=1225.473,90.881,-47.282,-178.563,5.548,148.541
C08281=1225.468,91.131,-47.300,-178.560,5.549,148.540
C08282=1225.464,91.380,-47.319,-178.558,5.550,148.540
C08283=1225.459,91.629,-47.337,-178.555,5.551,148.539
C08284=1225.453,91.878,-47.355,-178.553,5.552,148.538
C08285=1225.448,92.128,-47.373,-178.550,5.552,148.538
C08286=1225.444,92.377,-47.392,-178.548,5.553,148.537
C08287=1225.440,92.626,-47.410,-178.545,5.554,148.537
C08288=1225.434,92.876,-47.429,-178.543,5.554,148.536
C08289=1225.429,93.124,-47.448,-178.540,5.555,148.536
C08290=1225.425,93.374,-47.466,-178.537,5.557,148.535
C08291=1225.420,93.623,-47.484,-178.535,5.557,148.534
C08292=1225.414,93.873,-47.503,-178.532,5.558,148.534
C08293=1225.410,94.122,-47.522,-178.530,5.559,148.533
C08294=1225.405,94.371,-47.540,-178.527,5.559,148.533
C08295=1225.401,94.620,-47.558,-178.525,5.560,148.532
C08296=1225.396,94.870,-47.577,-178.522,5.562,148.532
C08297=1225.391,95.119,-47.595,-178.519,5.562,148.531
C08298=1225.386,95.368,-47.613,-178.517,5.563,148.530
C08299=1225.381,95.617,-47.632,-178.515,5.564,148.530
C08300=1225.376,95.867,-47.651,-178.512,5.565,148.529
C08301=1225.372,96.115,-47.669,-178.509,5.565,148.529
C08302=1225.366,96.365,-47.688,-178.507,5.566,148.528
C08303=1225.362,96.615,-47.706,-178.504,5.568,148.528
C08304=1225.357,96.863,-47.725,-178.501,5.568,148.527
C08305=1225.352,97.113,-47.744,-178.499,5.569,148.526
C08306=1225.348,97.362,-47.763,-178.497,5.570,148.526
C08307=1225.343,97.611,-47.781,-178.494,5.570,148.525
C08308=1225.338,97.861,-47.800,-178.491,5.572,148.525
C08309=1225.333,98.110,-47.818,-178.489,5.573,148.524
C08310=1225.328,98.359,-47.837,-178.486,5.573,148.523
C08311=1225.323,98.609,-47.856,-178.484,5.574,148.523
C08312=1225.318,98.858,-47.874,-178.481,5.575,148.522
C08313=1225.313,99.107,-47.893,-178.479,5.576,148.522
C08314=1225.309,99.357,-47.912,-178.476,5.577,148.521
C08315=1225.304,99.605,-47.930,-178.473,5.578,148.521
C08316=1225.299,99.855,-47.950,-178.471,5.579,148.520
C08317=1225.294,100.104,-47.968,-178.469,5.579,148.520
C08318=1225.289,100.353,-47.987,-178.466,5.580,148.519
C08319=1225.285,100.603,-48.006,-178.463,5.582,148.518
C08320=1225.280,100.851,-48.024,-178.461,5.582,148.518
C08321=1225.275,101.101,-48.043,-178.458,5.583,148.517
C08322=1225.271,101.350,-48.062,-178.455,5.584,148.517
C08323=1225.265,101.600,-48.080,-178.453,5.585,148.516
C08324=1225.261,101.849,-48.100,-178.450,5.586,148.516
C08325=1225.256,102.098,-48.119,-178.448,5.587,148.515
C08326=1225.251,102.348,-48.137,-178.445,5.588,148.515
C08327=1225.246,102.596,-48.156,-178.443,5.588,148.514
C08328=1225.241,102.845,-48.175,-178.440,5.589,148.513
C08329=1225.236,103.095,-48.194,-178.438,5.591,148.513
C08330=1225.232,103.344,-48.213,-178.435,5.591,148.512
C08331=1225.227,103.594,-48.232,-178.432,5.592,148.512
C08332=1225.222,103.842,-48.250,-178.430,5.593,148.511
C08333=1225.217,104.092,-48.270,-178.428,5.593,148.510
C08334=1225.213,104.341,-48.289,-178.425,5.595,148.510
C08335=1225.208,104.591,-48.308,-178.422,5.596,148.509
C08336=1225.203,104.839,-48.326,-178.420,5.596,148.509
C08337=1225.198,105.089,-48.346,-178.418,5.597,148.508
C08338=1225.193,105.338,-48.364,-178.415,5.598,148.508
C08339=1225.188,105.587,-48.383,-178.412,5.599,148.507
C08340=1225.183,105.836,-48.403,-178.410,5.600,148.507
C08341=1225.179,106.085,-48.422,-178.407,5.601,148.506
C08342=1225.174,106.335,-48.441,-178.404,5.602,148.505
C08343=1225.169,106.584,-48.459,-178.402,5.603,148.505
C08344=1225.164,106.833,-48.479,-178.399,5.604,148.504
C08345=1225.160,107.082,-48.498,-178.397,5.605,148.504
C08346=1225.154,107.351,-48.518,-178.394,5.606,148.503
C08347=1225.149,107.619,-48.539,-178.391,5.607,148.503
C08348=1225.144,107.888,-48.560,-178.389,5.608,148.502
C08349=1225.139,108.157,-48.580,-178.385,5.609,148.501
C08350=1225.134,108.406,-48.599,-178.383,5.610,148.501
C08351=1225.129,108.655,-48.619,-178.381,5.611,148.500
C08352=1225.124,108.904,-48.638,-178.378,5.611,148.500
C08353=1225.120,109.153,-48.657,-178.375,5.613,148.499
C08354=1225.115,109.402,-48.676,-178.373,5.614,148.499
C08355=1225.110,109.652,-48.696,-178.370,5.614,148.498
C08356=1225.105,109.901,-48.714,-178.368,5.615,148.498
C08357=1225.100,110.150,-48.734,-178.365,5.617,148.497
C08358=1225.095,110.399,-48.753,-178.363,5.618,148.497
C08359=1225.091,110.649,-48.772,-178.360,5.618,148.496
C08360=1225.086,110.897,-48.791,-178.357,5.619,148.495
C08361=1225.081,111.147,-48.811,-178.355,5.621,148.495
C08362=1225.077,111.396,-48.830,-178.352,5.621,148.494
C08363=1225.072,111.645,-48.849,-178.350,5.622,148.494
C08364=1225.067,111.895,-48.869,-178.347,5.623,148.493
C08365=1225.061,112.144,-48.888,-178.344,5.624,148.493
C08366=1225.057,112.393,-48.907,-178.342,5.625,148.492
C08367=1225.053,112.642,-48.927,-178.339,5.626,148.491
C08368=1225.047,112.891,-48.946,-178.337,5.627,148.491
C08369=1225.043,113.141,-48.966,-178.334,5.628,148.490
C08370=1225.038,113.389,-48.984,-178.332,5.629,148.490
C08371=1225.033,113.639,-49.004,-178.329,5.630,148.489
C08372=1225.029,113.889,-49.024,-178.327,5.631,148.489
C08373=1225.023,114.137,-49.043,-178.324,5.632,148.488
C08374=1225.019,114.387,-49.062,-178.322,5.633,148.488
C08375=1225.014,114.636,-49.081,-178.319,5.634,148.487
C08376=1225.009,114.885,-49.101,-178.317,5.634,148.487
C08377=1225.004,115.135,-49.121,-178.314,5.636,148.486
C08378=1224.999,115.384,-49.140,-178.312,5.637,148.486
C08379=1224.995,115.633,-49.159,-178.309,5.638,148.485
C08380=1224.991,115.882,-49.179,-178.306,5.639,148.484
C08381=1224.985,116.131,-49.199,-178.304,5.640,148.484
C08382=1224.980,116.380,-49.218,-178.301,5.641,148.483
C08383=1224.976,116.630,-49.238,-178.299,5.642,148.483
C08384=1224.970,116.879,-49.257,-178.296,5.643,148.482
C08385=1224.966,117.128,-49.276,-178.294,5.644,148.482
C08386=1224.961,117.377,-49.296,-178.291,5.645,148.481
C08387=1224.957,117.626,-49.316,-178.288,5.646,148.481
C08388=1224.952,117.875,-49.336,-178.286,5.647,148.480
C08389=1224.947,118.125,-49.355,-178.283,5.648,148.480
C08390=1224.942,118.374,-49.375,-178.281,5.649,148.479
C08391=1224.937,118.623,-49.394,-178.278,5.650,148.478
C08392=1224.933,118.872,-49.415,-178.276,5.651,148.478
C08393=1224.928,119.121,-49.433,-178.273,5.652,148.477
C08394=1224.923,119.370,-49.453,-178.270,5.653,148.477
C08395=1224.918,119.620,-49.473,-178.268,5.654,148.476
C08396=1224.913,119.868,-49.493,-178.265,5.655,148.476
C08397=1224.909,120.118,-49.512,-178.263,5.656,148.475
C08398=1224.904,120.367,-49.532,-178.260,5.657,148.475
C08399=1224.899,120.617,-49.552,-178.258,5.658,148.474
C08400=1224.894,120.865,-49.572,-178.255,5.659,148.474
C08401=1224.889,121.115,-49.591,-178.252,5.660,148.473
C08402=1224.885,121.364,-49.611,-178.250,5.661,148.473
C08403=1224.880,121.612,-49.631,-178.247,5.662,148.472
C08404=1224.875,121.862,-49.651,-178.245,5.663,148.472
C08405=1224.870,122.112,-49.670,-178.242,5.664,148.471
C08406=1224.866,122.361,-49.691,-178.240,5.665,148.471
C08407=1224.860,122.609,-49.710,-178.237,5.667,148.470
C08408=1224.856,122.859,-49.730,-178.235,5.668,148.470
C08409=1224.851,123.108,-49.750,-178.232,5.668,148.469
C08410=1224.846,123.358,-49.770,-178.229,5.670,148.469
C08411=1224.841,123.606,-49.790,-178.227,5.671,148.468
C08412=1224.837,123.855,-49.809,-178.224,5.671,148.467
C08413=1224.832,124.105,-49.829,-178.222,5.672,148.467
C08414=1224.827,124.354,-49.849,-178.219,5.674,148.466
C08415=1224.823,124.603,-49.869,-178.217,5.675,148.466
C08416=1224.818,124.852,-49.889,-178.214,5.675,148.465
C08417=1224.813,125.101,-49.909,-178.211,5.677,148.465
C08418=1224.809,125.350,-49.929,-178.209,5.678,148.464
C08419=1224.804,125.600,-49.949,-178.207,5.679,148.464
C08420=1224.799,125.849,-49.969,-178.203,5.680,148.463
C08421=1224.794,126.098,-49.988,-178.201,5.681,148.463
C08422=1224.790,126.347,-50.009,-178.199,5.682,148.462
C08423=1224.785,126.596,-50.028,-178.196,5.683,148.462
C08424=1224.780,126.845,-50.049,-178.193,5.684,148.461
C08425=1224.775,127.095,-50.069,-178.191,5.685,148.461
C08426=1224.770,127.344,-50.089,-178.188,5.687,148.460
C08427=1224.765,127.593,-50.109,-178.186,5.687,148.460
C08428=1224.761,127.842,-50.129,-178.183,5.689,148.459
C08429=1224.756,128.091,-50.149,-178.180,5.690,148.458
C08430=1224.752,128.340,-50.169,-178.178,5.691,148.458
C08431=1224.747,128.589,-50.189,-178.175,5.692,148.457
C08432=1224.742,128.839,-50.209,-178.173,5.693,148.457
C08433=1224.737,129.088,-50.230,-178.170,5.694,148.456
C08434=1224.732,129.337,-50.249,-178.168,5.695,148.456
C08435=1224.727,129.586,-50.270,-178.165,5.696,148.455
C08436=1224.723,129.835,-50.290,-178.163,5.697,148.455
C08437=1224.718,130.084,-50.310,-178.160,5.698,148.454
C08438=1224.714,130.333,-50.330,-178.158,5.699,148.454
C08439=1224.709,130.583,-50.351,-178.155,5.700,148.453
C08440=1224.704,130.832,-50.371,-178.152,5.702,148.453
C08441=1224.699,131.081,-50.391,-178.150,5.702,148.452
C08442=1224.694,131.329,-50.411,-178.147,5.704,148.452
C08443=1224.689,131.579,-50.431,-178.144,5.705,148.451
C08444=1224.684,131.828,-50.452,-178.142,5.706,148.451
C08445=1224.680,132.077,-50.472,-178.139,5.707,148.450
C08446=1224.675,132.327,-50.492,-178.137,5.708,148.450
C08447=1224.671,132.576,-50.512,-178.134,5.709,148.449
C08448=1224.666,132.825,-50.533,-178.132,5.711,148.449
C08449=1224.661,133.074,-50.554,-178.129,5.711,148.448
C08450=1224.656,133.343,-50.575,-178.127,5.713,148.448
C08451=1224.651,133.611,-50.597,-178.124,5.714,148.447
C08452=1224.645,133.880,-50.619,-178.121,5.715,148.447
C08453=1224.641,134.149,-50.641,-178.119,5.716,148.446
C08454=1224.636,134.398,-50.662,-178.115,5.718,148.446
C08455=1224.631,134.647,-50.681,-178.113,5.719,148.445
C08456=1224.626,134.896,-50.702,-178.110,5.720,148.444
C08457=1224.621,135.145,-50.722,-178.108,5.721,148.444
C08458=1224.617,135.394,-50.743,-178.106,5.722,148.443
C08459=1224.612,135.643,-50.764,-178.103,5.724,148.443
C08460=1224.607,135.892,-50.784,-178.100,5.724,148.442
C08461=1224.603,136.141,-50.805,-178.098,5.725,148.442
C08462=1224.597,136.391,-50.825,-178.095,5.727,148.441
C08463=1224.593,136.640,-50.845,-178.093,5.728,148.441
C08464=1224.588,136.889,-50.866,-178.090,5.729,148.440
C08465=1224.583,137.138,-50.887,-178.088,5.730,148.440
C08466=1224.579,137.387,-50.907,-178.085,5.731,148.439
C08467=1224.574,137.636,-50.927,-178.082,5.733,148.439
C08468=1224.569,137.885,-50.948,-178.080,5.734,148.439
C08469=1224.565,138.134,-50.969,-178.077,5.735,148.438
C08470=1224.559,138.383,-50.990,-178.075,5.736,148.438
C08471=1224.555,138.632,-51.010,-178.072,5.737,148.437
C08472=1224.551,138.881,-51.030,-178.070,5.738,148.437
C08473=1224.545,139.130,-51.051,-178.067,5.739,148.436
C08474=1224.541,139.379,-51.072,-178.064,5.741,148.436
C08475=1224.536,139.629,-51.093,-178.062,5.742,148.435
C08476=1224.531,139.878,-51.113,-178.059,5.743,148.435
C08477=1224.526,140.127,-51.134,-178.056,5.744,148.434
C08478=1224.522,140.376,-51.154,-178.054,5.745,148.434
C08479=1224.518,140.626,-51.175,-178.052,5.747,148.433
C08480=1224.513,140.875,-51.196,-178.049,5.747,148.433
C08481=1224.508,141.124,-51.216,-178.046,5.749,148.432
C08482=1224.503,141.373,-51.237,-178.044,5.750,148.432
C08483=1224.499,141.622,-51.258,-178.041,5.752,148.431
C08484=1224.494,141.871,-51.279,-178.039,5.752,148.431
C08485=1224.489,142.120,-51.299,-178.036,5.753,148.430
C08486=1224.484,142.369,-51.321,-178.033,5.755,148.430
C08487=1224.480,142.618,-51.341,-178.031,5.756,148.429
C08488=1224.475,142.867,-51.362,-178.029,5.758,148.429
C08489=1224.470,143.116,-51.382,-178.026,5.758,148.428
C08490=1224.465,143.365,-51.403,-178.023,5.760,148.428
C08491=1224.461,143.614,-51.424,-178.021,5.761,148.427
C08492=1224.456,143.864,-51.445,-178.019,5.762,148.427
C08493=1224.451,144.113,-51.467,-178.015,5.763,148.426
C08494=1224.447,144.362,-51.487,-178.013,5.764,148.426
C08495=1224.442,144.611,-51.508,-178.011,5.766,148.425
C08496=1224.437,144.860,-51.529,-178.008,5.766,148.425
C08497=1224.432,145.109,-51.549,-178.005,5.768,148.424
C08498=1224.428,145.357,-51.571,-178.003,5.769,148.424
C08499=1224.423,145.607,-51.592,-178.000,5.771,148.423
C08500=1224.419,145.856,-51.612,-177.997,5.771,148.423
C08501=1224.414,146.106,-51.633,-177.995,5.772,148.422
C08502=1224.409,146.354,-51.655,-177.993,5.774,148.422
C08503=1224.404,146.603,-51.675,-177.990,5.775,148.421
C08504=1224.399,146.853,-51.696,-177.987,5.777,148.421
C08505=1224.394,147.101,-51.718,-177.985,5.777,148.420
C08506=1224.390,147.351,-51.739,-177.982,5.779,148.420
C08507=1224.385,147.600,-51.760,-177.980,5.780,148.420
C08508=1224.381,147.849,-51.780,-177.977,5.782,148.419
C08509=1224.376,148.098,-51.802,-177.975,5.783,148.419
C08510=1224.371,148.347,-51.823,-177.972,5.784,148.418
C08511=1224.366,148.596,-51.843,-177.970,5.785,148.418
C08512=1224.362,148.845,-51.865,-177.967,5.787,148.417
C08513=1224.357,149.094,-51.886,-177.964,5.787,148.417
C08514=1224.352,149.343,-51.908,-177.962,5.789,148.416
C08515=1224.348,149.592,-51.928,-177.959,5.790,148.416
C08516=1224.342,149.841,-51.949,-177.957,5.791,148.415
C08517=1224.338,150.091,-51.971,-177.954,5.793,148.415
C08518=1224.334,150.340,-51.992,-177.952,5.793,148.414
C08519=1224.329,150.588,-52.013,-177.949,5.795,148.414
C08520=1224.324,150.837,-52.034,-177.946,5.796,148.413
C08521=1224.319,151.086,-52.056,-177.944,5.798,148.413
C08522=1224.315,151.336,-52.077,-177.942,5.799,148.412
C08523=1224.310,151.585,-52.098,-177.938,5.800,148.412
C08524=1224.305,151.834,-52.119,-177.936,5.801,148.411
C08525=1224.300,152.083,-52.140,-177.933,5.803,148.411
C08526=1224.296,152.332,-52.162,-177.931,5.804,148.410
C08527=1224.291,152.581,-52.183,-177.928,5.805,148.410
C08528=1224.286,152.830,-52.204,-177.926,5.806,148.409
C08529=1224.281,153.079,-52.226,-177.923,5.808,148.409
C08530=1224.277,153.328,-52.247,-177.921,5.809,148.409
C08531=1224.273,153.577,-52.268,-177.918,5.810,148.408
C08532=1224.267,153.826,-52.289,-177.916,5.811,148.408
C08533=1224.263,154.075,-52.311,-177.913,5.813,148.407
C08534=1224.258,154.325,-52.332,-177.911,5.814,148.407
C08535=1224.253,154.573,-52.354,-177.908,5.816,148.406
C08536=1224.249,154.822,-52.374,-177.905,5.816,148.406
C08537=1224.244,155.072,-52.396,-177.903,5.818,148.405
C08538=1224.240,155.320,-52.418,-177.901,5.819,148.405
C08539=1224.234,155.569,-52.439,-177.897,5.821,148.404
C08540=1224.229,155.818,-52.461,-177.895,5.822,148.404
C08541=1224.225,156.067,-52.483,-177.892,5.823,148.403
C08542=1224.220,156.317,-52.504,-177.890,5.824,148.403
C08543=1224.216,156.565,-52.525,-177.887,5.826,148.403
C08544=1224.212,156.814,-52.547,-177.885,5.826,148.402
C08545=1224.206,157.064,-52.568,-177.882,5.828,148.402
C08546=1224.202,157.312,-52.590,-177.879,5.830,148.401
C08547=1224.197,157.562,-52.612,-177.877,5.831,148.401
C08548=1224.192,157.811,-52.633,-177.874,5.833,148.400
C08549=1224.187,158.060,-52.654,-177.872,5.834,148.400
C08550=1224.183,158.309,-52.676,-177.869,5.835,148.399
C08551=1224.178,158.558,-52.698,-177.867,5.836,148.399
C08552=1224.173,158.807,-52.719,-177.864,5.838,148.398
C08553=1224.169,159.056,-52.741,-177.862,5.839,148.398
C08554=1224.164,159.325,-52.764,-177.859,5.840,148.397
C08555=1224.159,159.594,-52.788,-177.856,5.842,148.397
C08556=1224.154,159.863,-52.811,-177.854,5.843,148.396
C08557=1224.149,160.132,-52.835,-177.851,5.844,148.396
C08558=1224.144,160.381,-52.856,-177.848,5.846,148.395
C08559=1224.139,160.630,-52.878,-177.846,5.847,148.395
C08560=1224.135,160.879,-52.899,-177.843,5.849,148.394
C08561=1224.130,161.128,-52.921,-177.841,5.850,148.394
C08562=1224.125,161.377,-52.943,-177.838,5.851,148.394
C08563=1224.121,161.626,-52.965,-177.835,5.852,148.393
C08564=1224.116,161.876,-52.986,-177.833,5.854,148.393
C08565=1224.111,162.124,-53.008,-177.830,5.856,148.392
C08566=1224.107,162.374,-53.030,-177.827,5.856,148.392
C08567=1224.102,162.622,-53.052,-177.825,5.858,148.391
C08568=1224.097,162.871,-53.073,-177.823,5.859,148.391
C08569=1224.093,163.120,-53.095,-177.819,5.861,148.390
C08570=1224.088,163.369,-53.117,-177.817,5.862,148.390
C08571=1224.084,163.618,-53.139,-177.815,5.863,148.390
C08572=1224.079,163.867,-53.161,-177.812,5.864,148.389
C08573=1224.074,164.116,-53.183,-177.809,5.866,148.389
C08574=1224.069,164.365,-53.205,-177.807,5.868,148.388
C08575=1224.064,164.614,-53.227,-177.804,5.868,148.388
C08576=1224.060,164.863,-53.249,-177.802,5.870,148.387
C08577=1224.055,165.112,-53.270,-177.799,5.871,148.387
C08578=1224.051,165.361,-53.293,-177.796,5.873,148.386
C08579=1224.046,165.610,-53.314,-177.794,5.874,148.386
C08580=1224.042,165.859,-53.336,-177.792,5.876,148.386
C08581=1224.037,166.108,-53.358,-177.789,5.877,148.385
C08582=1224.032,166.357,-53.381,-177.786,5.878,148.385
C08583=1224.027,166.606,-53.402,-177.784,5.880,148.384
C08584=1224.022,166.855,-53.424,-177.782,5.881,148.384
C08585=1224.018,167.104,-53.446,-177.778,5.882,148.383
C08586=1224.013,167.353,-53.468,-177.776,5.884,148.383
C08587=1224.008,167.602,-53.490,-177.774,5.885,148.383
C08588=1224.004,167.851,-53.513,-177.771,5.887,148.382
C08589=1223.999,168.100,-53.535,-177.768,5.888,148.382
C08590=1223.995,168.349,-53.557,-177.766,5.890,148.381
C08591=1223.990,168.598,-53.578,-177.764,5.891,148.381
C08592=1223.986,168.847,-53.601,-177.761,5.892,148.380
C08593=1223.980,169.096,-53.623,-177.758,5.894,148.380
C08594=1223.976,169.345,-53.645,-177.756,5.895,148.379
C08595=1223.971,169.593,-53.667,-177.753,5.897,148.379
C08596=1223.967,169.843,-53.689,-177.751,5.897,148.378
C08597=1223.962,170.092,-53.712,-177.748,5.899,148.378
C08598=1223.957,170.341,-53.734,-177.745,5.901,148.378
C08599=1223.953,170.590,-53.756,-177.743,5.902,148.377
C08600=1223.948,170.838,-53.778,-177.740,5.903,148.377
C08601=1223.943,171.088,-53.801,-177.737,5.905,148.376
C08602=1223.938,171.336,-53.822,-177.735,5.906,148.376
C08603=1223.934,171.586,-53.844,-177.732,5.908,148.375
C08604=1223.929,171.834,-53.867,-177.730,5.909,148.375
C08605=1223.924,172.083,-53.889,-177.727,5.911,148.375
C08606=1223.920,172.333,-53.912,-177.725,5.912,148.374
C08607=1223.916,172.581,-53.934,-177.722,5.913,148.374
C08608=1223.911,172.831,-53.957,-177.719,5.915,148.373
C08609=1223.906,173.079,-53.978,-177.717,5.916,148.373
C08610=1223.902,173.328,-54.001,-177.715,5.918,148.373
C08611=1223.897,173.578,-54.024,-177.712,5.919,148.372
C08612=1223.892,173.826,-54.045,-177.709,5.920,148.372
C08613=1223.888,174.075,-54.068,-177.707,5.922,148.371
C08614=1223.882,174.324,-54.090,-177.704,5.924,148.371
C08615=1223.878,174.573,-54.112,-177.702,5.925,148.370
C08616=1223.873,174.822,-54.136,-177.699,5.926,148.370
C08617=1223.868,175.071,-54.157,-177.697,5.927,148.370
C08618=1223.864,175.320,-54.180,-177.694,5.929,148.369
C08619=1223.859,175.569,-54.203,-177.691,5.931,148.369
C08620=1223.855,175.817,-54.225,-177.689,5.932,148.368
C08621=1223.850,176.067,-54.248,-177.686,5.934,148.368
C08622=1223.846,176.316,-54.270,-177.684,5.935,148.368
C08623=1223.841,176.564,-54.292,-177.681,5.936,148.367
C08624=1223.836,176.814,-54.315,-177.678,5.938,148.367
C08625=1223.832,177.063,-54.338,-177.676,5.940,148.366
C08626=1223.827,177.312,-54.360,-177.674,5.941,148.366
C08627=1223.823,177.560,-54.383,-177.671,5.942,148.365
C08628=1223.818,177.810,-54.405,-177.668,5.944,148.365
C08629=1223.813,178.058,-54.428,-177.666,5.945,148.365
C08630=1223.808,178.308,-54.451,-177.663,5.947,148.364
C08631=1223.804,178.556,-54.473,-177.660,5.949,148.364
C08632=1223.799,178.805,-54.496,-177.658,5.949,148.363
C08633=1223.794,179.054,-54.518,-177.655,5.951,148.363
C08634=1223.790,179.303,-54.542,-177.653,5.953,148.363
C08635=1223.785,179.552,-54.563,-177.650,5.954,148.362
C08636=1223.780,179.801,-54.587,-177.647,5.956,148.362
C08637=1223.776,180.049,-54.609,-177.645,5.957,148.361
C08638=1223.771,180.299,-54.632,-177.643,5.958,148.361
C08639=1223.767,180.547,-54.655,-177.640,5.960,148.360
C08640=1223.762,180.797,-54.677,-177.637,5.962,148.360
C08641=1223.758,181.045,-54.700,-177.635,5.963,148.359
C08642=1223.753,181.295,-54.723,-177.632,5.965,148.359
C08643=1223.748,181.543,-54.745,-177.629,5.966,148.359
C08644=1223.743,181.792,-54.768,-177.627,5.967,148.358
C08645=1223.739,182.041,-54.791,-177.625,5.969,148.358
C08646=1223.735,182.290,-54.814,-177.622,5.971,148.357
C08647=1223.729,182.539,-54.837,-177.619,5.972,148.357
C08648=1223.725,182.788,-54.860,-177.617,5.974,148.357
C08649=1223.720,183.037,-54.883,-177.614,5.975,148.356
C08650=1223.716,183.286,-54.905,-177.612,5.976,148.356
C08651=1223.711,183.534,-54.928,-177.609,5.978,148.355
C08652=1223.706,183.783,-54.951,-177.606,5.980,148.355
C08653=1223.702,184.032,-54.974,-177.604,5.981,148.355
C08654=1223.698,184.281,-54.997,-177.602,5.983,148.354
C08655=1223.693,184.531,-55.020,-177.599,5.984,148.354
C08656=1223.688,184.779,-55.042,-177.596,5.986,148.353
C08657=1223.683,185.028,-55.066,-177.594,5.987,148.353
C08658=1223.679,185.297,-55.090,-177.591,5.989,148.353
C08659=1223.673,185.567,-55.115,-177.588,5.991,148.352
C08660=1223.668,185.837,-55.140,-177.585,5.992,148.352
C08661=1223.663,186.106,-55.165,-177.583,5.994,148.351
C08662=1223.659,186.355,-55.188,-177.580,5.996,148.351
C08663=1223.654,186.604,-55.211,-177.578,5.997,148.351
C08664=1223.649,186.853,-55.235,-177.575,5.998,148.350
C08665=1223.645,187.102,-55.258,-177.572,6.000,148.350
C08666=1223.641,187.351,-55.281,-177.570,6.001,148.349
C08667=1223.635,187.599,-55.304,-177.567,6.003,148.349
C08668=1223.631,187.848,-55.327,-177.565,6.005,148.349
C08669=1223.627,188.097,-55.350,-177.562,6.006,148.348
C08670=1223.622,188.346,-55.373,-177.559,6.007,148.348
C08671=1223.617,188.595,-55.397,-177.557,6.009,148.347
C08672=1223.613,188.844,-55.420,-177.554,6.011,148.347
C08673=1223.608,189.094,-55.442,-177.552,6.013,148.347
C08674=1223.603,189.342,-55.465,-177.549,6.014,148.346
C08675=1223.598,189.591,-55.489,-177.547,6.016,148.346
C08676=1223.594,189.839,-55.513,-177.544,6.017,148.345
C08677=1223.590,190.088,-55.535,-177.542,6.018,148.345
C08678=1223.585,190.337,-55.559,-177.539,6.020,148.345
C08679=1223.581,190.586,-55.582,-177.536,6.022,148.344
C08680=1223.576,190.835,-55.605,-177.534,6.024,148.344
C08681=1223.571,191.084,-55.629,-177.532,6.025,148.344
C08682=1223.567,191.333,-55.652,-177.529,6.027,148.343
C08683=1223.563,191.582,-55.675,-177.526,6.028,148.343
C08684=1223.557,191.830,-55.698,-177.523,6.030,148.342
C08685=1223.553,192.079,-55.721,-177.521,6.031,148.342
C08686=1223.548,192.328,-55.745,-177.518,6.033,148.342
C08687=1223.543,192.577,-55.768,-177.516,6.035,148.341
C08688=1223.539,192.826,-55.792,-177.513,6.037,148.341
C08689=1223.534,193.075,-55.815,-177.511,6.038,148.341
C08690=1223.530,193.324,-55.838,-177.508,6.039,148.340
C08691=1223.525,193.573,-55.862,-177.505,6.041,148.340
C08692=1223.521,193.822,-55.885,-177.503,6.043,148.339
C08693=1223.516,194.071,-55.908,-177.501,6.044,148.339
C08694=1223.512,194.319,-55.932,-177.498,6.046,148.339
C08695=1223.507,194.568,-55.956,-177.495,6.047,148.338
C08696=1223.502,194.817,-55.979,-177.493,6.049,148.338
C08697=1223.498,195.066,-56.002,-177.491,6.050,148.337
C08698=1223.493,195.315,-56.026,-177.487,6.052,148.337
C08699=1223.488,195.564,-56.050,-177.485,6.054,148.337
C08700=1223.484,195.813,-56.073,-177.482,6.055,148.336
C08701=1223.479,196.062,-56.097,-177.479,6.057,148.336
C08702=1223.475,196.310,-56.121,-177.477,6.058,148.335
C08703=1223.470,196.559,-56.144,-177.475,6.060,148.335
C08704=1223.465,196.808,-56.167,-177.472,6.062,148.335
C08705=1223.461,197.057,-56.191,-177.469,6.064,148.334
C08706=1223.456,197.306,-56.215,-177.467,6.065,148.334
C08707=1223.451,197.555,-56.238,-177.464,6.066,148.334
C08708=1223.447,197.803,-56.262,-177.462,6.068,148.333
C08709=1223.442,198.052,-56.286,-177.459,6.070,148.333
C08710=1223.438,198.301,-56.309,-177.456,6.072,148.332
C08711=1223.433,198.550,-56.333,-177.454,6.073,148.332
C08712=1223.429,198.799,-56.356,-177.452,6.075,148.332
C08713=1223.424,199.048,-56.380,-177.449,6.077,148.331
C08714=1223.419,199.296,-56.404,-177.446,6.078,148.331
C08715=1223.415,199.545,-56.427,-177.444,6.079,148.331
C08716=1223.410,199.793,-56.451,-177.442,6.081,148.330
C08717=1223.406,200.043,-56.475,-177.438,6.083,148.330
C08718=1223.401,200.291,-56.499,-177.436,6.085,148.329
C08719=1223.397,200.540,-56.522,-177.433,6.087,148.329
C08720=1223.393,200.789,-56.546,-177.431,6.088,148.329
C08721=1223.387,201.038,-56.570,-177.428,6.089,148.328
C08722=1223.383,201.287,-56.595,-177.426,6.091,148.328
C08723=1223.378,201.536,-56.618,-177.423,6.093,148.328
C08724=1223.374,201.784,-56.642,-177.421,6.095,148.327
C08725=1223.369,202.033,-56.665,-177.418,6.097,148.327
C08726=1223.365,202.282,-56.689,-177.416,6.098,148.327
C08727=1223.360,202.531,-56.713,-177.413,6.100,148.326
C08728=1223.355,202.779,-56.737,-177.411,6.102,148.326
C08729=1223.350,203.029,-56.761,-177.407,6.103,148.325
C08730=1223.346,203.278,-56.785,-177.405,6.105,148.325
C08731=1223.342,203.526,-56.809,-177.403,6.106,148.325
C08732=1223.337,203.775,-56.833,-177.400,6.108,148.324
C08733=1223.333,204.023,-56.857,-177.397,6.110,148.324
C08734=1223.327,204.273,-56.881,-177.395,6.111,148.324
C08735=1223.323,204.521,-56.905,-177.392,6.113,148.323
C08736=1223.319,204.770,-56.929,-177.390,6.115,148.323
C08737=1223.315,205.019,-56.953,-177.387,6.116,148.323
C08738=1223.310,205.268,-56.977,-177.385,6.118,148.322
C08739=1223.305,205.517,-57.001,-177.382,6.120,148.322
C08740=1223.300,205.766,-57.025,-177.380,6.122,148.322
C08741=1223.296,206.014,-57.049,-177.377,6.124,148.321
C08742=1223.292,206.262,-57.073,-177.374,6.125,148.321
C08743=1223.287,206.512,-57.097,-177.372,6.126,148.321
C08744=1223.282,206.761,-57.121,-177.370,6.128,148.320
C08745=1223.278,207.009,-57.145,-177.367,6.130,148.320
C08746=1223.273,207.258,-57.170,-177.364,6.132,148.320
C08747=1223.268,207.507,-57.193,-177.361,6.133,148.319
C08748=1223.264,207.756,-57.218,-177.359,6.135,148.319
C08749=1223.259,208.005,-57.242,-177.356,6.136,148.318
C08750=1223.255,208.253,-57.266,-177.354,6.138,148.318
C08751=1223.250,208.502,-57.291,-177.351,6.140,148.318
C08752=1223.246,208.751,-57.314,-177.349,6.142,148.317
C08753=1223.241,209.000,-57.339,-177.346,6.144,148.317
C08754=1223.237,209.249,-57.363,-177.343,6.146,148.317
C08755=1223.232,209.497,-57.388,-177.341,6.147,148.316
C08756=1223.227,209.746,-57.412,-177.339,6.148,148.316
C08757=1223.223,209.995,-57.436,-177.336,6.150,148.316
C08758=1223.218,210.244,-57.461,-177.333,6.152,148.315
C08759=1223.214,210.493,-57.484,-177.331,6.154,148.315
C08760=1223.209,210.741,-57.508,-177.328,6.156,148.315
C08761=1223.205,210.990,-57.533,-177.325,6.158,148.314
C08762=1223.200,211.261,-57.560,-177.323,6.160,148.314
C08763=1223.195,211.530,-57.586,-177.320,6.161,148.314
C08764=1223.190,211.801,-57.613,-177.317,6.163,148.313
C08765=1223.185,212.071,-57.639,-177.314,6.165,148.313
C08766=1223.181,212.320,-57.663,-177.312,6.167,148.312
C08767=1223.176,212.569,-57.688,-177.309,6.169,148.312
C08768=1223.171,212.818,-57.712,-177.306,6.170,148.312
C08769=1223.167,213.067,-57.737,-177.304,6.172,148.311
C08770=1223.162,213.315,-57.761,-177.301,6.174,148.311
C08771=1223.157,213.564,-57.786,-177.299,6.176,148.311
C08772=1223.153,213.813,-57.810,-177.296,6.178,148.310
C08773=1223.148,214.062,-57.835,-177.294,6.179,148.310
C08774=1223.144,214.310,-57.859,-177.291,6.181,148.310
C08775=1223.139,214.559,-57.884,-177.289,6.183,148.309
C08776=1223.135,214.808,-57.909,-177.286,6.184,148.309
C08777=1223.130,215.056,-57.934,-177.283,6.186,148.309
C08778=1223.126,215.305,-57.958,-177.281,6.188,148.308
C08779=1223.121,215.554,-57.983,-177.278,6.190,148.308
C08780=1223.117,215.803,-58.007,-177.275,6.192,148.308
C08781=1223.112,216.052,-58.032,-177.273,6.194,148.307
C08782=1223.108,216.300,-58.056,-177.270,6.196,148.307
C08783=1223.103,216.549,-58.080,-177.268,6.197,148.307
C08784=1223.099,216.798,-58.106,-177.265,6.198,148.306
C08785=1223.094,217.046,-58.130,-177.263,6.200,148.306
C08786=1223.089,217.295,-58.155,-177.260,6.202,148.306
C08787=1223.085,217.544,-58.179,-177.258,6.204,148.305
C08788=1223.080,217.793,-58.204,-177.255,6.206,148.305
C08789=1223.076,218.041,-58.229,-177.252,6.208,148.305
C08790=1223.071,218.290,-58.254,-177.250,6.210,148.304
C08791=1223.066,218.539,-58.279,-177.247,6.211,148.304
C08792=1223.063,218.788,-58.303,-177.244,6.213,148.304
C08793=1223.058,219.036,-58.328,-177.242,6.215,148.304
C08794=1223.053,219.285,-58.352,-177.240,6.216,148.303
C08795=1223.049,219.534,-58.378,-177.238,6.218,148.303
C08796=1223.044,219.783,-58.402,-177.235,6.220,148.303
C08797=1223.040,220.031,-58.427,-177.232,6.222,148.302
C08798=1223.035,220.280,-58.452,-177.230,6.224,148.302
C08799=1223.030,220.529,-58.477,-177.227,6.226,148.302
C08800=1223.026,220.777,-58.502,-177.224,6.228,148.301
C08801=1223.022,221.027,-58.527,-177.222,6.230,148.301
C08802=1223.017,221.275,-58.552,-177.219,6.231,148.301
C08803=1223.013,221.523,-58.576,-177.217,6.233,148.300
C08804=1223.008,221.772,-58.601,-177.214,6.235,148.300
C08805=1223.003,222.021,-58.627,-177.211,6.237,148.300
C08806=1222.999,222.270,-58.652,-177.209,6.239,148.299
C08807=1222.994,222.518,-58.676,-177.207,6.240,148.299
C08808=1222.990,222.767,-58.702,-177.204,6.242,148.299
C08809=1222.985,223.016,-58.726,-177.201,6.244,148.298
C08810=1222.981,223.265,-58.752,-177.199,6.245,148.298
C08811=1222.976,223.513,-58.776,-177.197,6.248,148.298
C08812=1222.972,223.762,-58.802,-177.194,6.249,148.298
C08813=1222.967,224.011,-58.827,-177.191,6.251,148.297
C08814=1222.963,224.259,-58.852,-177.189,6.253,148.297
C08815=1222.958,224.508,-58.876,-177.186,6.255,148.297
C08816=1222.954,224.757,-58.902,-177.183,6.257,148.296
C08817=1222.949,225.005,-58.927,-177.181,6.259,148.296
C08818=1222.945,225.254,-58.953,-177.178,6.261,148.296
C08819=1222.940,225.503,-58.977,-177.176,6.262,148.295
C08820=1222.936,225.751,-59.002,-177.173,6.264,148.295
C08821=1222.931,226.000,-59.027,-177.170,6.266,148.295
C08822=1222.927,226.249,-59.053,-177.168,6.268,148.294
C08823=1222.922,226.497,-59.078,-177.165,6.270,148.294
C08824=1222.917,226.747,-59.103,-177.163,6.271,148.294
C08825=1222.913,226.995,-59.129,-177.161,6.273,148.293
C08826=1222.908,227.244,-59.154,-177.158,6.275,148.293
C08827=1222.905,227.493,-59.179,-177.156,6.277,148.293
C08828=1222.900,227.741,-59.204,-177.153,6.279,148.293
C08829=1222.895,227.990,-59.229,-177.150,6.281,148.292
C08830=1222.890,228.238,-59.255,-177.148,6.282,148.292
C08831=1222.886,228.487,-59.280,-177.145,6.284,148.292
C08832=1222.881,228.736,-59.305,-177.142,6.286,148.291
C08833=1222.877,228.984,-59.331,-177.140,6.288,148.291
C08834=1222.873,229.233,-59.356,-177.138,6.290,148.291
C08835=1222.868,229.482,-59.381,-177.135,6.292,148.290
C08836=1222.863,229.731,-59.407,-177.132,6.294,148.290
C08837=1222.858,229.979,-59.432,-177.130,6.296,148.290
C08838=1222.855,230.227,-59.457,-177.127,6.298,148.289
C08839=1222.850,230.477,-59.482,-177.125,6.300,148.289
C08840=1222.846,230.725,-59.508,-177.122,6.301,148.289
C08841=1222.841,230.974,-59.534,-177.120,6.304,148.289
C08842=1222.837,231.222,-59.559,-177.117,6.305,148.288
C08843=1222.832,231.471,-59.585,-177.115,6.307,148.288
C08844=1222.828,231.720,-59.610,-177.112,6.309,148.288
C08845=1222.823,231.968,-59.635,-177.109,6.311,148.287
C08846=1222.819,232.217,-59.661,-177.107,6.313,148.287
C08847=1222.815,232.466,-59.687,-177.104,6.315,148.287
C08848=1222.810,232.714,-59.712,-177.102,6.317,148.287
C08849=1222.806,232.963,-59.738,-177.099,6.319,148.286
C08850=1222.801,233.212,-59.764,-177.097,6.321,148.286
C08851=1222.795,233.461,-59.789,-177.094,6.323,148.286
C08852=1222.791,233.709,-59.815,-177.092,6.324,148.285
C08853=1222.787,233.958,-59.840,-177.089,6.325,148.285
C08854=1222.782,234.206,-59.866,-177.087,6.328,148.285
C08855=1222.778,234.455,-59.891,-177.085,6.330,148.285
C08856=1222.774,234.704,-59.917,-177.082,6.331,148.284
C08857=1222.769,234.952,-59.943,-177.079,6.333,148.284
C08858=1222.765,235.201,-59.968,-177.077,6.335,148.284
C08859=1222.760,235.450,-59.994,-177.074,6.337,148.283
C08860=1222.756,235.698,-60.019,-177.072,6.339,148.283
C08861=1222.751,235.946,-60.045,-177.069,6.341,148.283
C08862=1222.746,236.196,-60.072,-177.067,6.343,148.283
C08863=1222.742,236.444,-60.097,-177.064,6.345,148.282
C08864=1222.737,236.693,-60.123,-177.061,6.347,148.282
C08865=1222.733,236.941,-60.148,-177.059,6.349,148.282
C08866=1222.728,237.213,-60.176,-177.056,6.351,148.281
C08867=1222.723,237.484,-60.205,-177.053,6.353,148.281
C08868=1222.719,237.756,-60.233,-177.050,6.355,148.281
C08869=1222.713,238.027,-60.261,-177.048,6.357,148.280
C08870=1222.710,238.275,-60.287,-177.045,6.360,148.280
C08871=1222.705,238.524,-60.313,-177.042,6.362,148.280
C08872=1222.700,238.773,-60.339,-177.040,6.364,148.280
C08873=1222.696,239.021,-60.365,-177.037,6.365,148.279
C08874=1222.691,239.270,-60.390,-177.035,6.367,148.279
C08875=1222.687,239.519,-60.416,-177.033,6.370,148.279
C08876=1222.682,239.768,-60.442,-177.030,6.371,148.279
C08877=1222.678,240.015,-60.469,-177.027,6.373,148.278
C08878=1222.673,240.264,-60.494,-177.025,6.375,148.278
C08879=1222.669,240.513,-60.520,-177.023,6.377,148.278
C08880=1222.664,240.762,-60.546,-177.020,6.379,148.278
C08881=1222.660,241.011,-60.572,-177.017,6.381,148.277
C08882=1222.655,241.258,-60.598,-177.015,6.383,148.277
C08883=1222.650,241.507,-60.625,-177.012,6.385,148.277
C08884=1222.646,241.756,-60.650,-177.010,6.387,148.277
C08885=1222.642,242.005,-60.676,-177.007,6.389,148.276
C08886=1222.638,242.253,-60.703,-177.005,6.391,148.276
C08887=1222.633,242.502,-60.729,-177.002,6.393,148.276
C08888=1222.628,242.750,-60.754,-176.999,6.395,148.275
C08889=1222.624,242.999,-60.781,-176.997,6.397,148.275
C08890=1222.619,243.248,-60.807,-176.995,6.399,148.275
C08891=1222.615,243.497,-60.833,-176.992,6.400,148.275
C08892=1222.611,243.745,-60.859,-176.989,6.402,148.274
C08893=1222.606,243.993,-60.885,-176.987,6.405,148.274
C08894=1222.602,244.242,-60.911,-176.985,6.406,148.274
C08895=1222.597,244.490,-60.938,-176.982,6.408,148.274
C08896=1222.593,244.739,-60.964,-176.979,6.410,148.273
C08897=1222.589,244.987,-60.990,-176.977,6.412,148.273
C08898=1222.584,245.237,-61.017,-176.975,6.414,148.273
C08899=1222.580,245.485,-61.042,-176.972,6.416,148.273
C08900=1222.575,245.734,-61.069,-176.969,6.418,148.272
C08901=1222.570,245.982,-61.095,-176.967,6.420,148.272
C08902=1222.566,246.230,-61.121,-176.965,6.422,148.272
C08903=1222.561,246.479,-61.148,-176.962,6.425,148.272
C08904=1222.557,246.727,-61.174,-176.959,6.427,148.271
C08905=1222.552,246.977,-61.200,-176.957,6.429,148.271
C08906=1222.548,247.225,-61.227,-176.954,6.431,148.271
C08907=1222.543,247.474,-61.253,-176.952,6.433,148.271
C08908=1222.539,247.722,-61.280,-176.949,6.434,148.270
C08909=1222.535,247.971,-61.305,-176.947,6.437,148.270
C08910=1222.531,248.219,-61.333,-176.944,6.438,148.270
C08911=1222.526,248.468,-61.358,-176.942,6.440,148.270
C08912=1222.521,248.716,-61.385,-176.939,6.443,148.270
C08913=1222.517,248.964,-61.411,-176.937,6.444,148.269
C08914=1222.512,249.213,-61.438,-176.934,6.446,148.269
C08915=1222.508,249.462,-61.465,-176.932,6.448,148.269
C08916=1222.503,249.711,-61.491,-176.929,6.450,148.269
C08917=1222.499,249.959,-61.518,-176.927,6.452,148.268
C08918=1222.495,250.207,-61.544,-176.924,6.455,148.268
C08919=1222.490,250.456,-61.570,-176.922,6.457,148.268
C08920=1222.486,250.705,-61.597,-176.919,6.459,148.268
C08921=1222.481,250.953,-61.624,-176.916,6.461,148.267
C08922=1222.477,251.202,-61.650,-176.914,6.463,148.267
C08923=1222.472,251.450,-61.677,-176.912,6.465,148.267
C08924=1222.468,251.699,-61.704,-176.909,6.467,148.267
C08925=1222.463,251.948,-61.730,-176.906,6.469,148.266
C08926=1222.459,252.196,-61.757,-176.904,6.471,148.266
C08927=1222.455,252.444,-61.783,-176.902,6.473,148.266
C08928=1222.450,252.693,-61.810,-176.899,6.475,148.266
C08929=1222.445,252.942,-61.837,-176.897,6.477,148.265
C08930=1222.441,253.190,-61.863,-176.894,6.480,148.265
C08931=1222.437,253.439,-61.890,-176.891,6.481,148.265
C08932=1222.433,253.687,-61.917,-176.889,6.484,148.265
C08933=1222.428,253.935,-61.944,-176.886,6.486,148.264
C08934=1222.423,254.184,-61.970,-176.884,6.487,148.264
C08935=1222.419,254.433,-61.996,-176.882,6.490,148.264
C08936=1222.415,254.681,-62.024,-176.879,6.491,148.264
C08937=1222.410,254.930,-62.051,-176.876,6.493,148.263
C08938=1222.406,255.178,-62.077,-176.874,6.496,148.263
C08939=1222.401,255.426,-62.104,-176.872,6.497,148.263
C08940=1222.397,255.675,-62.132,-176.868,6.500,148.263
C08941=1222.392,255.925,-62.158,-176.866,6.502,148.263
C08942=1222.388,256.173,-62.184,-176.864,6.504,148.262
C08943=1222.384,256.421,-62.211,-176.861,6.506,148.262
C08944=1222.379,256.670,-62.238,-176.859,6.508,148.262
C08945=1222.375,256.918,-62.265,-176.856,6.510,148.262
C08946=1222.371,257.166,-62.292,-176.854,6.512,148.261
C08947=1222.366,257.415,-62.319,-176.852,6.514,148.261
C08948=1222.361,257.663,-62.346,-176.849,6.517,148.261
C08949=1222.357,257.912,-62.373,-176.846,6.519,148.261
C08950=1222.353,258.160,-62.400,-176.844,6.521,148.261
C08951=1222.349,258.409,-62.427,-176.841,6.523,148.260
C08952=1222.344,258.658,-62.454,-176.839,6.525,148.260
C08953=1222.339,258.906,-62.481,-176.836,6.527,148.260
C08954=1222.335,259.154,-62.508,-176.834,6.529,148.260
C08955=1222.331,259.403,-62.535,-176.832,6.531,148.260
C08956=1222.326,259.651,-62.562,-176.829,6.534,148.259
C08957=1222.321,259.900,-62.589,-176.826,6.536,148.259
C08958=1222.317,260.148,-62.616,-176.824,6.538,148.259
C08959=1222.313,260.397,-62.644,-176.821,6.540,148.259
C08960=1222.309,260.645,-62.671,-176.819,6.542,148.259
C08961=1222.304,260.894,-62.698,-176.816,6.544,148.258
C08962=1222.300,261.142,-62.725,-176.814,6.546,148.258
C08963=1222.295,261.391,-62.752,-176.811,6.549,148.258
C08964=1222.290,261.639,-62.779,-176.809,6.551,148.258
C08965=1222.286,261.888,-62.806,-176.806,6.553,148.257
C08966=1222.282,262.136,-62.834,-176.804,6.555,148.257
C08967=1222.277,262.385,-62.861,-176.801,6.557,148.257
C08968=1222.273,262.633,-62.888,-176.799,6.559,148.257
C08969=1222.269,262.881,-62.915,-176.796,6.561,148.257
C08970=1222.264,263.154,-62.945,-176.793,6.563,148.256
C08971=1222.260,263.427,-62.975,-176.791,6.566,148.256
C08972=1222.254,263.700,-63.005,-176.788,6.568,148.256
C08973=1222.250,263.973,-63.034,-176.785,6.570,148.256
C08974=1222.245,264.220,-63.062,-176.783,6.573,148.256
C08975=1222.240,264.469,-63.089,-176.780,6.575,148.255
C08976=1222.236,264.718,-63.117,-176.778,6.577,148.255
C08977=1222.232,264.966,-63.144,-176.775,6.579,148.255
C08978=1222.227,265.215,-63.171,-176.773,6.581,148.255
C08979=1222.223,265.463,-63.198,-176.771,6.583,148.255
C08980=1222.218,265.711,-63.226,-176.767,6.586,148.254
C08981=1222.214,265.960,-63.254,-176.765,6.588,148.254
C08982=1222.210,266.209,-63.281,-176.763,6.590,148.254
C08983=1222.205,266.456,-63.308,-176.760,6.592,148.254
C08984=1222.201,266.705,-63.336,-176.758,6.594,148.254
C08985=1222.197,266.954,-63.364,-176.755,6.596,148.253
C08986=1222.192,267.202,-63.391,-176.753,6.599,148.253
C08987=1222.188,267.451,-63.418,-176.750,6.601,148.253
C08988=1222.183,267.699,-63.447,-176.748,6.603,148.253
C08989=1222.178,267.948,-63.474,-176.745,6.605,148.253
C08990=1222.174,268.196,-63.501,-176.743,6.607,148.253
C08991=1222.169,268.444,-63.528,-176.740,6.610,148.252
C08992=1222.166,268.693,-63.557,-176.738,6.612,148.252
C08993=1222.161,268.941,-63.584,-176.735,6.614,148.252
C08994=1222.157,269.189,-63.611,-176.733,6.616,148.252
C08995=1222.153,269.438,-63.639,-176.731,6.618,148.252
C08996=1222.148,269.686,-63.667,-176.728,6.621,148.251
C08997=1222.144,269.935,-63.694,-176.725,6.623,148.251
C08998=1222.139,270.184,-63.722,-176.723,6.625,148.251
C08999=1222.135,270.432,-63.749,-176.721,6.627,148.251
C09000=1222.130,270.680,-63.777,-176.718,6.629,148.251
C09001=1222.126,270.929,-63.805,-176.715,6.632,148.251
C09002=1222.122,271.177,-63.832,-176.713,6.634,148.250
C09003=1222.117,271.425,-63.860,-176.711,6.636,148.250
C09004=1222.113,271.675,-63.888,-176.708,6.638,148.250
C09005=1222.108,271.922,-63.916,-176.706,6.640,148.250
C09006=1222.104,272.171,-63.943,-176.703,6.643,148.250
C09007=1222.100,272.419,-63.971,-176.701,6.645,148.249
C09008=1222.096,272.667,-63.999,-176.698,6.647,148.249
C09009=1222.090,272.916,-64.027,-176.696,6.649,148.249
C09010=1222.086,273.165,-64.055,-176.693,6.651,148.249
C09011=1222.082,273.413,-64.083,-176.691,6.654,148.249
C09012=1222.078,273.661,-64.111,-176.688,6.656,148.248
C09013=1222.073,273.910,-64.138,-176.686,6.658,148.248
C09014=1222.069,274.158,-64.166,-176.684,6.661,148.248
C09015=1222.065,274.406,-64.194,-176.681,6.663,148.248
C09016=1222.060,274.655,-64.221,-176.679,6.665,148.248
C09017=1222.056,274.904,-64.250,-176.676,6.667,148.248
C09018=1222.051,275.152,-64.278,-176.674,6.670,148.248
C09019=1222.047,275.400,-64.306,-176.671,6.672,148.247
C09020=1222.042,275.648,-64.334,-176.669,6.674,148.247
C09021=1222.038,275.897,-64.361,-176.666,6.676,148.247
C09022=1222.034,276.146,-64.390,-176.664,6.679,148.247
C09023=1222.030,276.393,-64.417,-176.661,6.680,148.247
C09024=1222.025,276.642,-64.446,-176.659,6.684,148.247
C09025=1222.021,276.890,-64.474,-176.656,6.685,148.246
C09026=1222.017,277.139,-64.502,-176.654,6.688,148.246
C09027=1222.012,277.387,-64.530,-176.652,6.690,148.246
C09028=1222.007,277.635,-64.557,-176.649,6.693,148.246
C09029=1222.003,277.884,-64.586,-176.646,6.695,148.246
C09030=1221.999,278.132,-64.614,-176.644,6.697,148.246
C09031=1221.995,278.381,-64.642,-176.642,6.699,148.245
C09032=1221.990,278.629,-64.671,-176.639,6.702,148.245
C09033=1221.986,278.878,-64.699,-176.636,6.704,148.245
C09034=1221.982,279.125,-64.726,-176.634,6.706,148.245
C09035=1221.977,279.374,-64.755,-176.632,6.708,148.245
C09036=1221.973,279.622,-64.783,-176.629,6.711,148.245
C09037=1221.968,279.871,-64.812,-176.626,6.713,148.245
C09038=1221.964,280.119,-64.839,-176.624,6.715,148.244
C09039=1221.959,280.368,-64.868,-176.622,6.718,148.244
C09040=1221.955,280.616,-64.896,-176.619,6.720,148.244
C09041=1221.951,280.865,-64.925,-176.617,6.722,148.244
C09042=1221.946,281.112,-64.952,-176.614,6.724,148.244
C09043=1221.942,281.361,-64.981,-176.612,6.727,148.244
C09044=1221.938,281.610,-65.009,-176.610,6.729,148.244
C09045=1221.934,281.858,-65.037,-176.607,6.731,148.243
C09046=1221.929,282.107,-65.066,-176.605,6.733,148.243
C09047=1221.925,282.354,-65.094,-176.602,6.736,148.243
C09048=1221.921,282.603,-65.123,-176.600,6.738,148.243
C09049=1221.916,282.851,-65.151,-176.597,6.741,148.243
C09050=1221.912,283.100,-65.180,-176.595,6.742,148.243
C09051=1221.907,283.348,-65.208,-176.592,6.745,148.243
C09052=1221.903,283.596,-65.236,-176.590,6.748,148.243
C09053=1221.898,283.845,-65.265,-176.587,6.750,148.242
C09054=1221.894,284.093,-65.293,-176.585,6.753,148.242
C09055=1221.890,284.341,-65.322,-176.583,6.755,148.242
C09056=1221.886,284.589,-65.350,-176.580,6.757,148.242
C09057=1221.881,284.838,-65.379,-176.578,6.759,148.242
C09058=1221.876,285.086,-65.407,-176.575,6.762,148.242
C09059=1221.873,285.334,-65.436,-176.573,6.764,148.242
C09060=1221.868,285.583,-65.465,-176.571,6.766,148.241
C09061=1221.864,285.831,-65.492,-176.568,6.769,148.241
C09062=1221.860,286.079,-65.522,-176.565,6.771,148.241
C09063=1221.855,286.328,-65.551,-176.563,6.773,148.241
C09064=1221.851,286.576,-65.578,-176.560,6.776,148.241
C09065=1221.846,286.825,-65.607,-176.558,6.778,148.241
C09066=1221.841,287.073,-65.636,-176.556,6.780,148.241
C09067=1221.838,287.321,-65.664,-176.554,6.783,148.241
C09068=1221.833,287.570,-65.693,-176.551,6.785,148.240
C09069=1221.828,287.818,-65.722,-176.548,6.787,148.240
C09070=1221.825,288.066,-65.750,-176.546,6.790,148.240
C09071=1221.820,288.314,-65.780,-176.543,6.792,148.240
C09072=1221.815,288.563,-65.808,-176.541,6.795,148.240
C09073=1221.812,288.811,-65.836,-176.539,6.797,148.240
C09074=1221.807,289.085,-65.869,-176.536,6.800,148.240
C09075=1221.802,289.359,-65.900,-176.533,6.803,148.240
C09076=1221.798,289.634,-65.932,-176.531,6.805,148.240
C09077=1221.793,289.908,-65.964,-176.528,6.808,148.239
C09078=1221.788,290.156,-65.993,-176.526,6.810,148.239
C09079=1221.783,290.404,-66.021,-176.523,6.813,148.239
C09080=1221.779,290.653,-66.051,-176.520,6.815,148.239
C09081=1221.775,290.901,-66.079,-176.518,6.817,148.239
C09082=1221.771,291.149,-66.108,-176.516,6.820,148.239
C09083=1221.766,291.398,-66.137,-176.514,6.822,148.239
C09084=1221.761,291.645,-66.166,-176.511,6.824,148.239
C09085=1221.758,291.894,-66.194,-176.509,6.826,148.239
C09086=1221.754,292.142,-66.223,-176.506,6.829,148.238
C09087=1221.749,292.390,-66.253,-176.504,6.832,148.238
C09088=1221.744,292.639,-66.281,-176.501,6.833,148.238
C09089=1221.740,292.887,-66.311,-176.499,6.836,148.238
C09090=1221.736,293.135,-66.339,-176.497,6.839,148.238
C09091=1221.732,293.384,-66.368,-176.495,6.841,148.238
C09092=1221.727,293.631,-66.397,-176.492,6.844,148.238
C09093=1221.723,293.880,-66.426,-176.489,6.846,148.238
C09094=1221.719,294.128,-66.456,-176.487,6.848,148.238
C09095=1221.715,294.377,-66.485,-176.484,6.851,148.238
C09096=1221.710,294.626,-66.514,-176.482,6.853,148.238
C09097=1221.705,294.873,-66.543,-176.480,6.855,148.237
C09098=1221.702,295.121,-66.572,-176.477,6.858,148.237
C09099=1221.697,295.370,-66.600,-176.475,6.860,148.237
C09100=1221.693,295.618,-66.630,-176.473,6.863,148.237
C09101=1221.688,295.866,-66.659,-176.470,6.866,148.237
C09102=1221.684,296.114,-66.688,-176.468,6.868,148.237
C09103=1221.680,296.363,-66.717,-176.465,6.871,148.237
C09104=1221.676,296.611,-66.747,-176.463,6.873,148.237
C09105=1221.671,296.860,-66.776,-176.461,6.875,148.237
C09106=1221.667,297.108,-66.806,-176.458,6.878,148.237
C09107=1221.662,297.355,-66.835,-176.456,6.880,148.237
C09108=1221.658,297.604,-66.863,-176.454,6.883,148.237
C09109=1221.654,297.853,-66.893,-176.451,6.885,148.236
C09110=1221.650,298.101,-66.922,-176.449,6.887,148.236
C09111=1221.645,298.349,-66.952,-176.446,6.890,148.236
C09112=1221.641,298.597,-66.981,-176.444,6.893,148.236
C09113=1221.636,298.845,-67.010,-176.442,6.895,148.236
C09114=1221.632,299.093,-67.040,-176.440,6.897,148.236
C09115=1221.628,299.341,-67.069,-176.437,6.900,148.236
C09116=1221.624,299.590,-67.098,-176.434,6.902,148.236
C09117=1221.619,299.839,-67.127,-176.432,6.904,148.236
C09118=1221.615,300.087,-67.157,-176.430,6.907,148.236
C09119=1221.611,300.335,-67.186,-176.427,6.910,148.236
C09120=1221.606,300.583,-67.215,-176.425,6.913,148.236
C09121=1221.602,300.831,-67.245,-176.423,6.915,148.236
C09122=1221.598,301.079,-67.274,-176.421,6.917,148.236
C09123=1221.594,301.327,-67.304,-176.418,6.920,148.236
C09124=1221.589,301.576,-67.333,-176.416,6.922,148.236
C09125=1221.585,301.824,-67.363,-176.413,6.924,148.235
C09126=1221.581,302.072,-67.392,-176.411,6.927,148.235
C09127=1221.576,302.321,-67.422,-176.408,6.929,148.235
C09128=1221.572,302.569,-67.452,-176.406,6.933,148.235
